METHOD FB_init : BOOL
VAR_INPUT
	bInitRetains : BOOL; // if TRUE, the retain variables are initialized (warm start / cold start)
	bInCopyCode : BOOL;  // if TRUE, the instance afterwards gets moved into the copy code (online change)
END_VAR
AddInput('aPoint1', aPoint1);
AddInput('aPoint2', aPoint2);
AddParameter('bNormalize', bNormalize);
AddInput('hrPrev', hrPrev);
AddOutput('aDirection', aDirection);
AddOutput('hresult',hresult);
END_METHOD

METHOD PUBLIC  Clone : I_Node
VAR
	pNode : POINTER TO Node_F_VN_PointToPointDirection_TcVnPoint2_DINT;
END_VAR
pNode := __NEW(Node_F_VN_PointToPointDirection_TcVnPoint2_DINT);
Clone := pNode^;
END_METHOD

METHOD PROTECTED OnExecute
hresult.Value := F_VN_PointToPointDirection_TcVnPoint2_DINT(
    aPoint1 := aPoint1.Value,
    aPoint2 := aPoint2.Value,
    aDirection := aDirection.Value,
    bNormalize := bNormalize.Value,
	hrPrev:= hrPrev.Value);
END_METHOD

METHOD PUBLIC PreExecutionCheck
VAR_INPUT
	Check : I_PreExecutionChecks;
END_VAR
END_METHOD

END_FUNCTION_BLOCK

// Nodes/Miscellaneous/Node_F_VN_PointToPointDirection_TcVnPoint2_LREAL
{attribute 'linkalways'} 
{attribute 'no_explicit_call' := 'This FB is a CLASS and must be accessed using methods or properties'}
{attribute 'enable_dynamic_creation'}
FUNCTION_BLOCK Node_F_VN_PointToPointDirection_TcVnPoint2_LREAL EXTENDS VisionNode
VAR
    aPoint1 : _TcVnPoint2_LREAL;
    aPoint2 : _TcVnPoint2_LREAL;
    aDirection : _TcVnVector2_LREAL;
    bNormalize : _BOOL(FALSE);
    hrPrev : _HRESULT(S_OK);
	hresult : _HRESULT(S_OK);
END_VAR

METHOD FB_init : BOOL
VAR_INPUT
	bInitRetains : BOOL; // if TRUE, the retain variables are initialized (warm start / cold start)
	bInCopyCode : BOOL;  // if TRUE, the instance afterwards gets moved into the copy code (online change)
END_VAR
AddInput('aPoint1', aPoint1);
AddInput('aPoint2', aPoint2);
AddParameter('bNormalize', bNormalize);
AddInput('hrPrev', hrPrev);
AddOutput('aDirection', aDirection);
AddOutput('hresult',hresult);
END_METHOD

METHOD PUBLIC  Clone : I_Node
VAR
	pNode : POINTER TO Node_F_VN_PointToPointDirection_TcVnPoint2_LREAL;
END_VAR
pNode := __NEW(Node_F_VN_PointToPointDirection_TcVnPoint2_LREAL);
Clone := pNode^;
END_METHOD

METHOD PROTECTED OnExecute
hresult.Value := F_VN_PointToPointDirection_TcVnPoint2_LREAL(
    aPoint1 := aPoint1.Value,
    aPoint2 := aPoint2.Value,
    aDirection := aDirection.Value,
    bNormalize := bNormalize.Value,
	hrPrev:= hrPrev.Value);
END_METHOD

METHOD PUBLIC PreExecutionCheck
VAR_INPUT
	Check : I_PreExecutionChecks;
END_VAR
END_METHOD

END_FUNCTION_BLOCK

// Nodes/Miscellaneous/Node_F_VN_PointToPointDirection_TcVnPoint2_REAL
{attribute 'linkalways'} 
{attribute 'no_explicit_call' := 'This FB is a CLASS and must be accessed using methods or properties'}
{attribute 'enable_dynamic_creation'}
FUNCTION_BLOCK Node_F_VN_PointToPointDirection_TcVnPoint2_REAL EXTENDS VisionNode
VAR
    aPoint1 : _TcVnPoint2_REAL;
    aPoint2 : _TcVnPoint2_REAL;
    aDirection : _TcVnVector2_REAL;
    bNormalize : _BOOL(FALSE);
    hrPrev : _HRESULT(S_OK);
	hresult : _HRESULT(S_OK);
END_VAR

METHOD FB_init : BOOL
VAR_INPUT
	bInitRetains : BOOL; // if TRUE, the retain variables are initialized (warm start / cold start)
	bInCopyCode : BOOL;  // if TRUE, the instance afterwards gets moved into the copy code (online change)
END_VAR
AddInput('aPoint1', aPoint1);
AddInput('aPoint2', aPoint2);
AddParameter('bNormalize', bNormalize);
AddInput('hrPrev', hrPrev);
AddOutput('aDirection', aDirection);
AddOutput('hresult',hresult);
END_METHOD

METHOD PUBLIC  Clone : I_Node
VAR
	pNode : POINTER TO Node_F_VN_PointToPointDirection_TcVnPoint2_REAL;
END_VAR
pNode := __NEW(Node_F_VN_PointToPointDirection_TcVnPoint2_REAL);
Clone := pNode^;
END_METHOD

METHOD PROTECTED OnExecute
hresult.Value := F_VN_PointToPointDirection_TcVnPoint2_REAL(
    aPoint1 := aPoint1.Value,
    aPoint2 := aPoint2.Value,
    aDirection := aDirection.Value,
    bNormalize := bNormalize.Value,
	hrPrev:= hrPrev.Value);
END_METHOD

METHOD PUBLIC PreExecutionCheck
VAR_INPUT
	Check : I_PreExecutionChecks;
END_VAR
END_METHOD

END_FUNCTION_BLOCK

// Nodes/Miscellaneous/Node_F_VN_PointToPointDistance_TcVnPoint2_DINT
{attribute 'linkalways'} 
{attribute 'no_explicit_call' := 'This FB is a CLASS and must be accessed using methods or properties'}
{attribute 'enable_dynamic_creation'}
FUNCTION_BLOCK Node_F_VN_PointToPointDistance_TcVnPoint2_DINT EXTENDS VisionNode
VAR
    aPoint1 : _TcVnPoint2_DINT;
    aPoint2 : _TcVnPoint2_DINT;
    fDistance : _LREAL(0.0);
    hrPrev : _HRESULT(S_OK);
	hresult : _HRESULT(S_OK);
END_VAR

METHOD FB_init : BOOL
VAR_INPUT
	bInitRetains : BOOL; // if TRUE, the retain variables are initialized (warm start / cold start)
	bInCopyCode : BOOL;  // if TRUE, the instance afterwards gets moved into the copy code (online change)
END_VAR
AddInput('aPoint1', aPoint1);
AddInput('aPoint2', aPoint2);
AddInput('hrPrev', hrPrev);
AddOutput('fDistance', fDistance);
AddOutput('hresult',hresult);
END_METHOD

METHOD PUBLIC  Clone : I_Node
VAR
	pNode : POINTER TO Node_F_VN_PointToPointDistance_TcVnPoint2_DINT;
END_VAR
pNode := __NEW(Node_F_VN_PointToPointDistance_TcVnPoint2_DINT);
Clone := pNode^;
END_METHOD

METHOD PROTECTED OnExecute
hresult.Value := F_VN_PointToPointDistance_TcVnPoint2_DINT(
    aPoint1 := aPoint1.Value,
    aPoint2 := aPoint2.Value,
    fDistance := fDistance.Value,
	hrPrev:= hrPrev.Value);
END_METHOD

METHOD PUBLIC PreExecutionCheck
VAR_INPUT
	Check : I_PreExecutionChecks;
END_VAR
END_METHOD

END_FUNCTION_BLOCK

// Nodes/Miscellaneous/Node_F_VN_PointToPointDistance_TcVnPoint2_LREAL
{attribute 'linkalways'} 
{attribute 'no_explicit_call' := 'This FB is a CLASS and must be accessed using methods or properties'}
{attribute 'enable_dynamic_creation'}
FUNCTION_BLOCK Node_F_VN_PointToPointDistance_TcVnPoint2_LREAL EXTENDS VisionNode
VAR
    aPoint1 : _TcVnPoint2_LREAL;
    aPoint2 : _TcVnPoint2_LREAL;
    fDistance : _LREAL(0.0);
    hrPrev : _HRESULT(S_OK);
	hresult : _HRESULT(S_OK);
END_VAR

METHOD FB_init : BOOL
VAR_INPUT
	bInitRetains : BOOL; // if TRUE, the retain variables are initialized (warm start / cold start)
	bInCopyCode : BOOL;  // if TRUE, the instance afterwards gets moved into the copy code (online change)
END_VAR
AddInput('aPoint1', aPoint1);
AddInput('aPoint2', aPoint2);
AddInput('hrPrev', hrPrev);
AddOutput('fDistance', fDistance);
AddOutput('hresult',hresult);
END_METHOD

METHOD PUBLIC  Clone : I_Node
VAR
	pNode : POINTER TO Node_F_VN_PointToPointDistance_TcVnPoint2_LREAL;
END_VAR
pNode := __NEW(Node_F_VN_PointToPointDistance_TcVnPoint2_LREAL);
Clone := pNode^;
END_METHOD

METHOD PROTECTED OnExecute
hresult.Value := F_VN_PointToPointDistance_TcVnPoint2_LREAL(
    aPoint1 := aPoint1.Value,
    aPoint2 := aPoint2.Value,
    fDistance := fDistance.Value,
	hrPrev:= hrPrev.Value);
END_METHOD

METHOD PUBLIC PreExecutionCheck
VAR_INPUT
	Check : I_PreExecutionChecks;
END_VAR
END_METHOD

END_FUNCTION_BLOCK

// Nodes/Miscellaneous/Node_F_VN_PointToPointDistance_TcVnPoint2_REAL
{attribute 'linkalways'} 
{attribute 'no_explicit_call' := 'This FB is a CLASS and must be accessed using methods or properties'}
{attribute 'enable_dynamic_creation'}
FUNCTION_BLOCK Node_F_VN_PointToPointDistance_TcVnPoint2_REAL EXTENDS VisionNode
VAR
    aPoint1 : _TcVnPoint2_REAL;
    aPoint2 : _TcVnPoint2_REAL;
    fDistance : _LREAL(0.0);
    hrPrev : _HRESULT(S_OK);
	hresult : _HRESULT(S_OK);
END_VAR

METHOD FB_init : BOOL
VAR_INPUT
	bInitRetains : BOOL; // if TRUE, the retain variables are initialized (warm start / cold start)
	bInCopyCode : BOOL;  // if TRUE, the instance afterwards gets moved into the copy code (online change)
END_VAR
AddInput('aPoint1', aPoint1);
AddInput('aPoint2', aPoint2);
AddInput('hrPrev', hrPrev);
AddOutput('fDistance', fDistance);
AddOutput('hresult',hresult);
END_METHOD

METHOD PUBLIC  Clone : I_Node
VAR
	pNode : POINTER TO Node_F_VN_PointToPointDistance_TcVnPoint2_REAL;
END_VAR
pNode := __NEW(Node_F_VN_PointToPointDistance_TcVnPoint2_REAL);
Clone := pNode^;
END_METHOD

METHOD PROTECTED OnExecute
hresult.Value := F_VN_PointToPointDistance_TcVnPoint2_REAL(
    aPoint1 := aPoint1.Value,
    aPoint2 := aPoint2.Value,
    fDistance := fDistance.Value,
	hrPrev:= hrPrev.Value);
END_METHOD

METHOD PUBLIC PreExecutionCheck
VAR_INPUT
	Check : I_PreExecutionChecks;
END_VAR
END_METHOD

END_FUNCTION_BLOCK

// Nodes/Miscellaneous/Node_F_VN_RotatedRectangleCorners
{attribute 'linkalways'} 
{attribute 'no_explicit_call' := 'This FB is a CLASS and must be accessed using methods or properties'}
{attribute 'enable_dynamic_creation'}
FUNCTION_BLOCK Node_F_VN_RotatedRectangleCorners EXTENDS VisionNode
VAR
    stRect : _TcVnRotatedRectangle;
    aCorners : _TcVnArray4_Point2_REAL;
    hrPrev : _HRESULT(S_OK);
	hresult : _HRESULT(S_OK);
END_VAR

METHOD FB_init : BOOL
VAR_INPUT
	bInitRetains : BOOL; // if TRUE, the retain variables are initialized (warm start / cold start)
	bInCopyCode : BOOL;  // if TRUE, the instance afterwards gets moved into the copy code (online change)
END_VAR
AddInput('stRect', stRect);
AddInput('hrPrev', hrPrev);
AddOutput('aCorners', aCorners);
AddOutput('hresult',hresult);
END_METHOD

METHOD PUBLIC  Clone : I_Node
VAR
	pNode : POINTER TO Node_F_VN_RotatedRectangleCorners;
END_VAR
pNode := __NEW(Node_F_VN_RotatedRectangleCorners);
Clone := pNode^;
END_METHOD

METHOD PROTECTED OnExecute
hresult.Value := F_VN_RotatedRectangleCorners(
    stRect := stRect.Value,
    aCorners := aCorners.Value,
	hrPrev:= hrPrev.Value);
END_METHOD

METHOD PUBLIC PreExecutionCheck
VAR_INPUT
	Check : I_PreExecutionChecks;
END_VAR
END_METHOD

END_FUNCTION_BLOCK

// Nodes/Miscellaneous/Node_F_VN_RotatedRectangleIntersection
{attribute 'linkalways'} 
{attribute 'no_explicit_call' := 'This FB is a CLASS and must be accessed using methods or properties'}
{attribute 'enable_dynamic_creation'}
FUNCTION_BLOCK Node_F_VN_RotatedRectangleIntersection EXTENDS VisionNode
VAR
    stRect1 : _TcVnRotatedRectangle;
    stRect2 : _TcVnRotatedRectangle;
    ipIntersection : _ITcVnContainer;
    eIntersection : _ETcVnRectangleIntersection(ETcVnRectangleIntersection.TCVN_RI_NONE);
    hrPrev : _HRESULT(S_OK);
	hresult : _HRESULT(S_OK);
END_VAR

METHOD FB_init : BOOL
VAR_INPUT
	bInitRetains : BOOL; // if TRUE, the retain variables are initialized (warm start / cold start)
	bInCopyCode : BOOL;  // if TRUE, the instance afterwards gets moved into the copy code (online change)
END_VAR
AddInput('stRect1', stRect1);
AddInput('stRect2', stRect2);
AddInput('hrPrev', hrPrev);
AddOutput('ipIntersection', ipIntersection);
AddOutput('eIntersection', eIntersection);
AddOutput('hresult',hresult);
END_METHOD

METHOD PUBLIC  Clone : I_Node
VAR
	pNode : POINTER TO Node_F_VN_RotatedRectangleIntersection;
END_VAR
pNode := __NEW(Node_F_VN_RotatedRectangleIntersection);
Clone := pNode^;
END_METHOD

METHOD PROTECTED OnExecute
VAR
    intersection : ETcVnRectangleIntersection;
END_VAR
hresult.Value := F_VN_RotatedRectangleIntersection(
    stRect1 := stRect1.Value,
    stRect2 := stRect2.Value,
    ipIntersection := ipIntersection.Value,
    eIntersection := intersection,
	hrPrev:= hrPrev.Value);

 eIntersection.Value := intersection;
END_METHOD

METHOD PUBLIC PreExecutionCheck
VAR_INPUT
	Check : I_PreExecutionChecks;
END_VAR
END_METHOD

END_FUNCTION_BLOCK

// Nodes/Neural Network/Node_F_VN_Reduce
{attribute 'linkalways'} 
{attribute 'no_explicit_call' := 'This FB is a CLASS and must be accessed using methods or properties'}
{attribute 'enable_dynamic_creation'}
FUNCTION_BLOCK Node_F_VN_Reduce EXTENDS VisionNode
VAR
    ipSrcImage : _ITcVnImage;
    ipDestImage : _ITcVnImage;
	nDim : _DINT(0);
	eReduceType : _ETcVnReduceType(ETcVnReduceType.TCVN_RT_REDUCE_AVG);
    hrPrev : _HRESULT(S_OK);
	hresult : _HRESULT(S_OK);
END_VAR

METHOD FB_init : BOOL
VAR_INPUT
	bInitRetains : BOOL; // if TRUE, the retain variables are initialized (warm start / cold start)
	bInCopyCode : BOOL;  // if TRUE, the instance afterwards gets moved into the copy code (online change)
END_VAR
AddInput('ipSrcImage', ipSrcImage);
AddInput('hrPrev', hrPrev);
AddParameter('nDim', nDim);
AddParameter('eReduceType', eReduceType);
AddOutput('ipDestImage', ipDestImage);
AddOutput('hresult',hresult);
END_METHOD

METHOD PUBLIC  Clone : I_Node
VAR
	pNode : POINTER TO Node_F_VN_Reduce;
END_VAR
pNode := __NEW(Node_F_VN_Reduce);
Clone := pNode^;
END_METHOD

METHOD PROTECTED OnExecute
hresult.Value := F_VN_Reduce(
	ipSrcImage := ipSrcImage.Value,
	ipDestImage := ipDestImage.Value,
	nDim := nDim.Value,
	eReduceType := eReduceType.Value,
	hrPrev:= hrPrev.Value);
END_METHOD

METHOD PUBLIC PreExecutionCheck
VAR_INPUT
	Check : I_PreExecutionChecks;
END_VAR
VAR
	nDimValue : DINT;
END_VAR
Check.IsTrue(ipSrcImage.IsValid, 'ipSrcImage must contain an image');
Check.IsTrue(ipSrcImage.HasChannelCount(1), 'ipSrcImage must have 1 channel');
Check.IsTrue(ipSrcImage.IsElementType(ETcVnElementType.TCVN_ET_USINT) OR_ELSE ipSrcImage.IsElementType(ETcVnElementType.TCVN_ET_REAL), 'ipSrcImage must have 32 bit pixel depth');

nDimValue := nDim.Value;
Check.IsTrue(nDimValue = 0 OR_ELSE nDimValue = 1 OR_ELSE nDimValue = 2, 'nDim must be 0, 1 or 2');
END_METHOD

END_FUNCTION_BLOCK

// Nodes/Neural Network/Node_F_VN_ReduceArg
{attribute 'linkalways'} 
{attribute 'no_explicit_call' := 'This FB is a CLASS and must be accessed using methods or properties'}
{attribute 'enable_dynamic_creation'}
FUNCTION_BLOCK Node_F_VN_ReduceArg EXTENDS VisionNode
VAR
    ipSrcImage : _ITcVnImage;
    ipDestImage : _ITcVnImage;
	nDim : _DINT(0);
	eReduceType : _DINT(0);
    hrPrev : _HRESULT(S_OK);
	hresult : _HRESULT(S_OK);
END_VAR

METHOD FB_init : BOOL
VAR_INPUT
	bInitRetains : BOOL; // if TRUE, the retain variables are initialized (warm start / cold start)
	bInCopyCode : BOOL;  // if TRUE, the instance afterwards gets moved into the copy code (online change)
END_VAR
AddInput('ipSrcImage', ipSrcImage);
AddInput('hrPrev', hrPrev);
AddParameter('nDim', nDim);
AddParameter('eReduceType', eReduceType);
AddOutput('ipDestImage', ipDestImage);
AddOutput('hresult',hresult);
END_METHOD

METHOD PUBLIC  Clone : I_Node
VAR
	pNode : POINTER TO Node_F_VN_ReduceArg;
END_VAR
pNode := __NEW(Node_F_VN_ReduceArg);
Clone := pNode^;
END_METHOD

METHOD PROTECTED OnExecute
hresult.Value := F_VN_ReduceArg(
	ipSrcImage := ipSrcImage.Value,
	ipDestImage := ipDestImage.Value,
	nDim := nDim.Value,
	eReduceType := eReduceType.Value,
	hrPrev:= hrPrev.Value);
END_METHOD

METHOD PUBLIC PreExecutionCheck
VAR_INPUT
	Check : I_PreExecutionChecks;
END_VAR
VAR
	nDimValue : DINT;
END_VAR
Check.IsTrue(ipSrcImage.IsValid, 'ipSrcImage must contain an image');
// Check.IsTrue(ipSrcImage.HasChannelCount(1), 'ipSrcImage must have 1 channel');
// Check.IsTrue(ipSrcImage.IsElementType(ETcVnElementType.TCVN_ET_USINT) OR_ELSE ipSrcImage.IsElementType(ETcVnElementType.TCVN_ET_REAL), 'ipSrcImage must have 32 bit pixel depth');

nDimValue := nDim.Value;
Check.IsTrue(nDimValue = 0 OR_ELSE nDimValue = 1 OR_ELSE nDimValue = 2, 'nDim must be 0, 1 or 2');
END_METHOD

END_FUNCTION_BLOCK

// Nodes/Neural Network/Node_F_VN_Sigmoid
{attribute 'linkalways'} 
{attribute 'no_explicit_call' := 'This FB is a CLASS and must be accessed using methods or properties'}
{attribute 'enable_dynamic_creation'}
FUNCTION_BLOCK Node_F_VN_Sigmoid EXTENDS VisionNode
VAR
    ipSrcImage : _ITcVnImage;
    ipDestImage : _ITcVnImage;
    hrPrev : _HRESULT(S_OK);
	hresult : _HRESULT(S_OK);
END_VAR

METHOD FB_init : BOOL
VAR_INPUT
	bInitRetains : BOOL; // if TRUE, the retain variables are initialized (warm start / cold start)
	bInCopyCode : BOOL;  // if TRUE, the instance afterwards gets moved into the copy code (online change)
END_VAR
AddInput('ipSrcImage', ipSrcImage);
AddInput('hrPrev', hrPrev);
AddOutput('ipDestImage', ipDestImage);
AddOutput('hresult',hresult);
END_METHOD

METHOD PUBLIC  Clone : I_Node
VAR
	pNode : POINTER TO Node_F_VN_Sigmoid;
END_VAR
pNode := __NEW(Node_F_VN_Sigmoid);
Clone := pNode^;
END_METHOD

METHOD PROTECTED OnExecute
hresult.Value := F_VN_Sigmoid(
    ipSrcImage := ipSrcImage.Value,
	ipDestImage := ipDestImage.Value,
	hrPrev:= hrPrev.Value);
END_METHOD

METHOD PUBLIC PreExecutionCheck
VAR_INPUT
	Check : I_PreExecutionChecks;
END_VAR
Check.IsTrue(ipSrcImage.IsValid, 'ipSrcImage must contain an image');
Check.IsTrue(ipSrcImage.IsElementType(ETcVnElementType.TCVN_ET_REAL), 'ipSrcImage must be element type REAL');
END_METHOD

END_FUNCTION_BLOCK

// Nodes/Neural Network/Node_F_VN_SigmoidExp
{attribute 'linkalways'} 
{attribute 'no_explicit_call' := 'This FB is a CLASS and must be accessed using methods or properties'}
{attribute 'enable_dynamic_creation'}
FUNCTION_BLOCK Node_F_VN_SigmoidExp EXTENDS VisionNode
VAR
    ipSrcImage : _ITcVnImage;
    ipDestImage : _ITcVnImage;
    fShift : _REAL(0.0);
    fSteepness : _REAL(0.0);
    hrPrev : _HRESULT(S_OK);
	hresult : _HRESULT(S_OK);
END_VAR

METHOD FB_init : BOOL
VAR_INPUT
	bInitRetains : BOOL; // if TRUE, the retain variables are initialized (warm start / cold start)
	bInCopyCode : BOOL;  // if TRUE, the instance afterwards gets moved into the copy code (online change)
END_VAR
AddInput('ipSrcImage', ipSrcImage);
AddParameter('fShift', fShift);
AddParameter('fSteepness', fSteepness);
AddInput('hrPrev', hrPrev);
AddOutput('ipDestImage', ipDestImage);
AddOutput('hresult',hresult);
END_METHOD

METHOD PUBLIC  Clone : I_Node
VAR
	pNode : POINTER TO Node_F_VN_SigmoidExp;
END_VAR
pNode := __NEW(Node_F_VN_SigmoidExp);
Clone := pNode^;
END_METHOD

METHOD PROTECTED OnExecute
hresult.Value := F_VN_SigmoidExp(
    ipSrcImage := ipSrcImage.Value,
	ipDestImage := ipDestImage.Value,
    fShift := fShift.Value,
    fSteepness := fSteepness.Value,
	hrPrev:= hrPrev.Value);
END_METHOD

METHOD PUBLIC PreExecutionCheck
VAR_INPUT
	Check : I_PreExecutionChecks;
END_VAR
Check.IsTrue(ipSrcImage.IsValid, 'ipSrcImage must contain an image');
Check.IsTrue(ipSrcImage.IsElementType(ETcVnElementType.TCVN_ET_REAL), 'ipSrcImage must be element type REAL');
END_METHOD

END_FUNCTION_BLOCK

// Nodes/Neural Network/Node_F_VN_SoftMax
{attribute 'linkalways'} 
{attribute 'no_explicit_call' := 'This FB is a CLASS and must be accessed using methods or properties'}
{attribute 'enable_dynamic_creation'}
FUNCTION_BLOCK Node_F_VN_SoftMax EXTENDS VisionNode
VAR
    ipSrcImage : _ITcVnImage;
    ipDestImage : _ITcVnImage;
    bFlatten : _BOOL(FALSE);
    hrPrev : _HRESULT(S_OK);
	hresult : _HRESULT(S_OK);
END_VAR

METHOD FB_init : BOOL
VAR_INPUT
	bInitRetains : BOOL; // if TRUE, the retain variables are initialized (warm start / cold start)
	bInCopyCode : BOOL;  // if TRUE, the instance afterwards gets moved into the copy code (online change)
END_VAR
AddInput('ipSrcImage', ipSrcImage);
AddParameter('bFlatten', bFlatten);
AddInput('hrPrev', hrPrev);
AddOutput('ipDestImage', ipDestImage);
AddOutput('hresult',hresult);
END_METHOD

METHOD PUBLIC  Clone : I_Node
VAR
	pNode : POINTER TO Node_F_VN_SoftMax;
END_VAR
pNode := __NEW(Node_F_VN_SoftMax);
Clone := pNode^;
END_METHOD

METHOD PROTECTED OnExecute
hresult.Value := F_VN_SoftMax(
    ipSrcImage := ipSrcImage.Value,
	ipDestImage := ipDestImage.Value,
    bFlatten := bFlatten.Value,
	hrPrev:= hrPrev.Value);
END_METHOD

METHOD PUBLIC PreExecutionCheck
VAR_INPUT
	Check : I_PreExecutionChecks;
END_VAR
Check.IsTrue(ipSrcImage.IsValid, 'ipSrcImage must contain an image');
Check.IsTrue(ipSrcImage.IsElementType(ETcVnElementType.TCVN_ET_REAL), 'ipSrcImage must be element type REAL');
Check.IsTrue(ipSrcImage.HasChannelCount(1), 'ipSrcImage must have 1 channel');
END_METHOD

END_FUNCTION_BLOCK

// Nodes/OCR/Node_F_VN_OCR
{attribute 'linkalways'} 
{attribute 'no_explicit_call' := 'This FB is a CLASS and must be accessed using methods or properties'}
{attribute 'enable_dynamic_creation'}
FUNCTION_BLOCK Node_F_VN_OCR EXTENDS VisionNode
VAR
	ipSrcImage : _ITcVnImage;
    eModel : _ETcVnOcrModelType(ETcVnOcrModelType.TCVN_OMT_NUMBERS);
    ipCharacters : _ITcVnContainer;
    hrPrev : _HRESULT(S_OK);
	hresult : _HRESULT(S_OK);
END_VAR

METHOD FB_init : BOOL
VAR_INPUT
	bInitRetains : BOOL; // if TRUE, the retain variables are initialized (warm start / cold start)
	bInCopyCode : BOOL;  // if TRUE, the instance afterwards gets moved into the copy code (online change)
END_VAR
AddInput('ipSrcImage', ipSrcImage);
AddParameter('eModel', eModel);
AddInput('hrPrev', hrPrev);
AddOutput('ipCharacters', ipCharacters);
AddOutput('hresult',hresult);
END_METHOD

METHOD PUBLIC  Clone : I_Node
VAR
	pNode : POINTER TO Node_F_VN_OCR;
END_VAR
pNode := __NEW(Node_F_VN_OCR);
Clone := pNode^;
END_METHOD

METHOD PROTECTED OnExecute
hresult.Value := F_VN_OCR(
	ipSrcImage := ipSrcImage.Value,
    eModel := eModel.Value,
	ipCharacters := ipCharacters.Value,
	hrPrev:= hrPrev.Value);
END_METHOD

METHOD PUBLIC PreExecutionCheck
VAR_INPUT
	Check : I_PreExecutionChecks;
END_VAR
VAR
    result : HRESULT;
END_VAR
result := F_VN_CheckFunctionInitialization(ETcVnInitializableFunction.TCVN_IF_OCR, eModel.Value, S_OK);
Check.IsTrue((result = S_OK), 'Invalid OCR model');

Check.IsTrue(ipSrcImage.IsValid, 'ipSrcImage must contain an image');
Check.IsTrue(ipSrcImage.IsPixelDepth(8), 'ipSrcImage must have 8 bit pixel depth');
Check.IsTrue(ipSrcImage.HasChannelCount(1), 'ipSrcImage must contain 1 channel');
END_METHOD

END_FUNCTION_BLOCK

// Nodes/OCR/Node_F_VN_OCRExp
{attribute 'linkalways'} 
{attribute 'no_explicit_call' := 'This FB is a CLASS and must be accessed using methods or properties'}
{attribute 'enable_dynamic_creation'}
FUNCTION_BLOCK Node_F_VN_OCRExp EXTENDS VisionNode
VAR
	ipSrcImage : _ITcVnImage;
    eModel : _ETcVnOcrModelType(ETcVnOcrModelType.TCVN_OMT_NUMBERS);
    ipCharacters : _ITcVnContainer;
    sPattern : _STRING('');
    eOcrOptions : _ETcVnOcrOptions(ETcVnOcrOptions.TCVN_OO_NONE);
    ipBoundingBoxes : _ITcVnContainer;
    ipConfidences : _ITcVnContainer;
    hrPrev : _HRESULT(S_OK);
    fMinConfidence : _REAL(0.0);
	hresult : _HRESULT(S_OK);
END_VAR

METHOD FB_init : BOOL
VAR_INPUT
	bInitRetains : BOOL; // if TRUE, the retain variables are initialized (warm start / cold start)
	bInCopyCode : BOOL;  // if TRUE, the instance afterwards gets moved into the copy code (online change)
END_VAR
AddInput('ipSrcImage', ipSrcImage);
AddParameter('eModel', eModel);
AddParameter('sPattern', sPattern);
AddParameter('eOcrOptions', eOcrOptions);
AddInput('hrPrev', hrPrev);
AddOutput('ipCharacters', ipCharacters);
AddOutput('ipBoundingBoxes', ipBoundingBoxes);
AddOutput('ipConfidences', ipConfidences);
AddOutput('fMinConfidence', fMinConfidence);
AddOutput('hresult',hresult);
END_METHOD

METHOD PUBLIC  Clone : I_Node
VAR
	pNode : POINTER TO Node_F_VN_OCRExp;
END_VAR
pNode := __NEW(Node_F_VN_OCRExp);
Clone := pNode^;
END_METHOD

METHOD PROTECTED OnExecute
VAR
    minConfidence : REAL;
END_VAR
hresult.Value := F_VN_OCRExp(
	ipSrcImage := ipSrcImage.Value,
    eModel := eModel.Value,
	ipCharacters := ipCharacters.Value,
    sPattern := sPattern.Value,
    eOcrOptions := eOcrOptions.Value,
    ipBoundingBoxes := ipBoundingBoxes.Value,
    ipConfidences := ipConfidences.Value,
	hrPrev := hrPrev.Value,
    fMinConfidence => minConfidence);

fMinConfidence.Value := minConfidence;
END_METHOD

METHOD PUBLIC PreExecutionCheck
VAR_INPUT
	Check : I_PreExecutionChecks;
END_VAR
VAR
    result : HRESULT;
END_VAR
result := F_VN_CheckFunctionInitialization(ETcVnInitializableFunction.TCVN_IF_OCR, eModel.Value, S_OK);
Check.IsTrue((result = S_OK), 'Invalid OCR model');

Check.IsTrue(ipSrcImage.IsValid, 'ipSrcImage must contain an image');
Check.IsTrue(ipSrcImage.IsPixelDepth(8), 'ipSrcImage must have 8 bit pixel depth');
Check.IsTrue(ipSrcImage.HasChannelCount(1), 'ipSrcImage must contain 1 channel');
END_METHOD

END_FUNCTION_BLOCK

// Nodes/Polarization/Node_F_VN_AngleAndDegreeOfLinearPolarization
{attribute 'linkalways'}
{attribute 'no_explicit_call' := 'This FB is a CLASS and must be accessed using methods or properties'}
{attribute 'enable_dynamic_creation'}
FUNCTION_BLOCK Node_F_VN_AngleAndDegreeOfLinearPolarization EXTENDS VisionNode
VAR
    ip0Deg : _ITcVnImage;
    ip45Deg : _ITcVnImage;
    ip90Deg : _ITcVnImage;
    ip135Deg : _ITcVnImage;
    ipAoLP : _ITcVnImage;
    ipDoLP : _ITcVnImage;
    eDestType : _ETcVnElementType(ETcVnElementType.TCVN_ET_REAL);
    hrPrev : _HRESULT(S_OK);
    hresult : _HRESULT(S_OK);
END_VAR

METHOD FB_init : BOOL
VAR_INPUT
    bInitRetains : BOOL;
    bInCopyCode : BOOL;
END_VAR
AddInput('ip0Deg', ip0Deg);
AddInput('ip45Deg', ip45Deg);
AddInput('ip90Deg', ip90Deg);
AddInput('ip135Deg', ip135Deg);
AddOutput('ipAoLP', ipAoLP);
AddOutput('ipDoLP', ipDoLP);
AddParameter('eDestType', eDestType);
AddInput('hrPrev', hrPrev);
AddOutput('hresult', hresult);
END_METHOD

METHOD PUBLIC Clone : I_Node
VAR
    pNode : POINTER TO Node_F_VN_AngleAndDegreeOfLinearPolarization;
END_VAR
pNode := __NEW(Node_F_VN_AngleAndDegreeOfLinearPolarization);
Clone := pNode^;
END_METHOD

METHOD PROTECTED OnExecute
hresult.Value := F_VN_AngleAndDegreeOfLinearPolarization(
    ip0Deg := ip0Deg.Value,
    ip45Deg := ip45Deg.Value,
    ip90Deg := ip90Deg.Value,
    ip135Deg := ip135Deg.Value,
    ipAoLP := ipAoLP.Value,
    ipDoLP := ipDoLP.Value,
    eDestType := eDestType.Value,
    hrPrev := hrPrev.Value);
END_METHOD

METHOD PUBLIC PreExecutionCheck
VAR_INPUT
    Check : I_PreExecutionChecks;
END_VAR
Check.IsTrue(ip0Deg.IsValid, 'ip0Deg must contain an image');
Check.IsTrue(ip0Deg.IsElementType(ETcVnElementType.TCVN_ET_USINT) OR
             ip0Deg.IsElementType(ETcVnElementType.TCVN_ET_UINT), 'Polarization components must contain USINT or UINT elements');
Check.IsTrue(ip0Deg.HasChannelCount(1) OR ip0Deg.HasChannelCount(3), 'Polarization components must contain 1 or 3 channels');
Check.IsTrue(ip45Deg.IsValid, 'ip45Deg must contain an image');
Check.IsTrue(ImagesHaveMatchingPixelFormats(ip0Deg.Value, ip45Deg.Value), 'Source images must have matching pixel formats');
Check.IsTrue(IsImage1SizeEqualToImage2Size(ip0Deg.Value, ip45Deg.Value), 'Source images must have matching dimensions');
Check.IsTrue(ip90Deg.IsValid, 'ip90Deg must contain an image');
Check.IsTrue(ImagesHaveMatchingPixelFormats(ip0Deg.Value, ip90Deg.Value), 'Source images must have matching pixel formats');
Check.IsTrue(IsImage1SizeEqualToImage2Size(ip0Deg.Value, ip90Deg.Value), 'Source images must have matching dimensions');
Check.IsTrue(ip135Deg.IsValid, 'ip135Deg must contain an image');
Check.IsTrue(ImagesHaveMatchingPixelFormats(ip0Deg.Value, ip135Deg.Value), 'Source images must have matching pixel formats');
Check.IsTrue(IsImage1SizeEqualToImage2Size(ip0Deg.Value, ip135Deg.Value), 'Source images must have matching dimensions');
Check.IsTrue((eDestType.Value = ETcVnElementType.TCVN_ET_REAL) OR
             (eDestType.Value = ETcVnElementType.TCVN_ET_USINT), 'Unsupported eDestType');
Check.IsTrue((ipAoLP.Value = 0) OR ((ipAoLP.Value <> ip0Deg.Value) AND
             (ipAoLP.Value <> ip45Deg.Value) AND
             (ipAoLP.Value <> ip90Deg.Value) AND
             (ipAoLP.Value <> ip135Deg.Value)), 'ipAoLP must be different from the source images');
Check.IsTrue((ipDoLP.Value = 0) OR ((ipDoLP.Value <> ip0Deg.Value) AND
             (ipDoLP.Value <> ip45Deg.Value) AND
             (ipDoLP.Value <> ip90Deg.Value) AND
             (ipDoLP.Value <> ip135Deg.Value)), 'ipDoLP must be different from the source images');
END_METHOD

END_FUNCTION_BLOCK

// Nodes/Polarization/Node_F_VN_DemosaicPolarizedImage
{attribute 'linkalways'}
{attribute 'no_explicit_call' := 'This FB is a CLASS and must be accessed using methods or properties'}
{attribute 'enable_dynamic_creation'}
FUNCTION_BLOCK Node_F_VN_DemosaicPolarizedImage EXTENDS VisionNode
VAR
    ipPolarizedImage : _ITcVnImage;
    ip0Deg : _ITcVnImage;
    ip45Deg : _ITcVnImage;
    ip90Deg : _ITcVnImage;
    ip135Deg : _ITcVnImage;
    eEncoding : _ETcVnPixelEncoding(ETcVnPixelEncoding.TCVN_PE_NONE);
    eInterpolation : _ETcVnPolarizedImageInterpolation(ETcVnPolarizedImageInterpolation.TCVN_PII_NONE);
    hrPrev : _HRESULT(S_OK);
    hresult : _HRESULT(S_OK);
END_VAR

METHOD FB_init : BOOL
VAR_INPUT
    bInitRetains : BOOL;
    bInCopyCode : BOOL;
END_VAR
AddInput('ipPolarizedImage', ipPolarizedImage);
AddOutput('ip0Deg', ip0Deg);
AddOutput('ip45Deg', ip45Deg);
AddOutput('ip90Deg', ip90Deg);
AddOutput('ip135Deg', ip135Deg);
AddParameter('eEncoding', eEncoding);
AddParameter('eInterpolation', eInterpolation);
AddInput('hrPrev', hrPrev);
AddOutput('hresult', hresult);
END_METHOD

METHOD PUBLIC Clone : I_Node
VAR
    pNode : POINTER TO Node_F_VN_DemosaicPolarizedImage;
END_VAR
pNode := __NEW(Node_F_VN_DemosaicPolarizedImage);
Clone := pNode^;
END_METHOD

METHOD PROTECTED OnExecute
hresult.Value := F_VN_DemosaicPolarizedImage(
    ipPolarizedImage := ipPolarizedImage.Value,
    ip0Deg := ip0Deg.Value,
    ip45Deg := ip45Deg.Value,
    ip90Deg := ip90Deg.Value,
    ip135Deg := ip135Deg.Value,
    eEncoding := eEncoding.Value,
    eInterpolation := eInterpolation.Value,
    hrPrev := hrPrev.Value);
END_METHOD

METHOD PUBLIC PreExecutionCheck
VAR_INPUT
    Check : I_PreExecutionChecks;
END_VAR
Check.IsTrue(ipPolarizedImage.IsValid, 'ipPolarizedImage must contain an image');
Check.IsTrue(ipPolarizedImage.IsElementType(ETcVnElementType.TCVN_ET_USINT) OR
             ipPolarizedImage.IsElementType(ETcVnElementType.TCVN_ET_UINT), 'Polarized image must contain USINT or UINT elements');
Check.IsTrue((eEncoding.Value = ETcVnPixelEncoding.TCVN_PE_NONE) OR
             (eEncoding.Value = ETcVnPixelEncoding.TCVN_PE_BAYER_GR) OR
             (eEncoding.Value = ETcVnPixelEncoding.TCVN_PE_BAYER_RG) OR
             (eEncoding.Value = ETcVnPixelEncoding.TCVN_PE_BAYER_GB) OR
             (eEncoding.Value = ETcVnPixelEncoding.TCVN_PE_BAYER_BG), 'Unsupported eEncoding');
Check.IsTrue((eInterpolation.Value = ETcVnPolarizedImageInterpolation.TCVN_PII_NONE) OR
             (eInterpolation.Value = ETcVnPolarizedImageInterpolation.TCVN_PII_NEAREST_NEIGHBOR) OR
             (eInterpolation.Value = ETcVnPolarizedImageInterpolation.TCVN_PII_BILINEAR) OR
             (eInterpolation.Value = ETcVnPolarizedImageInterpolation.TCVN_PII_BICUBIC) OR
             (eInterpolation.Value = ETcVnPolarizedImageInterpolation.TCVN_PII_LANCZOS4), 'Unsupported eInterpolation');
Check.IsTrue((ip0Deg.Value = 0) OR (ip0Deg.Value <> ipPolarizedImage.Value), 'ip0Deg must be different from the source image');
Check.IsTrue((ip45Deg.Value = 0) OR (ip45Deg.Value <> ipPolarizedImage.Value), 'ip45Deg must be different from the source image');
Check.IsTrue((ip90Deg.Value = 0) OR (ip90Deg.Value <> ipPolarizedImage.Value), 'ip90Deg must be different from the source image');
Check.IsTrue((ip135Deg.Value = 0) OR (ip135Deg.Value <> ipPolarizedImage.Value), 'ip135Deg must be different from the source image');
END_METHOD

END_FUNCTION_BLOCK

// Nodes/Polarization/Node_F_VN_PolarizedImageGlareReduction
{attribute 'linkalways'}
{attribute 'no_explicit_call' := 'This FB is a CLASS and must be accessed using methods or properties'}
{attribute 'enable_dynamic_creation'}
FUNCTION_BLOCK Node_F_VN_PolarizedImageGlareReduction EXTENDS VisionNode
VAR
    ipPolarizedImage : _ITcVnImage;
    ipDestImage : _ITcVnImage;
    eEncoding : _ETcVnPixelEncoding(ETcVnPixelEncoding.TCVN_PE_NONE);
    fIndex : _REAL(0.0);
    hrPrev : _HRESULT(S_OK);
    hresult : _HRESULT(S_OK);
END_VAR

METHOD FB_init : BOOL
VAR_INPUT
    bInitRetains : BOOL;
    bInCopyCode : BOOL;
END_VAR
AddInput('ipPolarizedImage', ipPolarizedImage);
AddOutput('ipDestImage', ipDestImage);
AddParameter('eEncoding', eEncoding);
AddParameter('fIndex', fIndex);
AddInput('hrPrev', hrPrev);
AddOutput('hresult', hresult);
END_METHOD

METHOD PUBLIC Clone : I_Node
VAR
    pNode : POINTER TO Node_F_VN_PolarizedImageGlareReduction;
END_VAR
pNode := __NEW(Node_F_VN_PolarizedImageGlareReduction);
Clone := pNode^;
END_METHOD

METHOD PROTECTED OnExecute
hresult.Value := F_VN_PolarizedImageGlareReduction(
    ipPolarizedImage := ipPolarizedImage.Value,
    ipDestImage := ipDestImage.Value,
    eEncoding := eEncoding.Value,
    fIndex := fIndex.Value,
    hrPrev := hrPrev.Value);
END_METHOD

METHOD PUBLIC PreExecutionCheck
VAR_INPUT
    Check : I_PreExecutionChecks;
END_VAR
Check.IsTrue(ipPolarizedImage.IsValid, 'ipPolarizedImage must contain an image');
Check.IsTrue(ipPolarizedImage.IsElementType(ETcVnElementType.TCVN_ET_USINT) OR
             ipPolarizedImage.IsElementType(ETcVnElementType.TCVN_ET_UINT), 'Polarized image must contain USINT or UINT elements');
Check.IsTrue((eEncoding.Value = ETcVnPixelEncoding.TCVN_PE_NONE) OR
             (eEncoding.Value = ETcVnPixelEncoding.TCVN_PE_BAYER_GR) OR
             (eEncoding.Value = ETcVnPixelEncoding.TCVN_PE_BAYER_RG) OR
             (eEncoding.Value = ETcVnPixelEncoding.TCVN_PE_BAYER_GB) OR
             (eEncoding.Value = ETcVnPixelEncoding.TCVN_PE_BAYER_BG), 'Unsupported eEncoding');
Check.IsTrue((fIndex.Value >= 0.0) AND (fIndex.Value <= 3.0), 'Intensity index must be between 0 and 3');
END_METHOD

END_FUNCTION_BLOCK

// Nodes/Texture Analysis/Node_F_VN_Granulometry
{attribute 'linkalways'} 
{attribute 'no_explicit_call' := 'This FB is a CLASS and must be accessed using methods or properties'}
{attribute 'enable_dynamic_creation'}
FUNCTION_BLOCK Node_F_VN_Granulometry EXTENDS VisionNode
VAR
    ipImage : _ITcVnImage;
    ipIntensityDiffs : _ITcVnContainer;
    eMorphType : _ETcVnMorphologicalOperator(ETcVnMorphologicalOperator.TCVN_MO_CLOSING);
    nMinSize : _UDINT(3);
    nMaxSize : _UDINT(3);
    nStep : _UDINT(2);
    hrPrev : _HRESULT(S_OK);
	hresult : _HRESULT(S_OK);
END_VAR

METHOD FB_init : BOOL
VAR_INPUT
	bInitRetains : BOOL; // if TRUE, the retain variables are initialized (warm start / cold start)
	bInCopyCode : BOOL;  // if TRUE, the instance afterwards gets moved into the copy code (online change)
END_VAR
AddInput('ipImage', ipImage);
AddParameter('eMorphType', eMorphType);
AddParameter('nMinSize', nMinSize);
AddParameter('nMaxSize', nMaxSize);
AddParameter('nStep', nStep);
AddInput('hrPrev', hrPrev);
AddOutput('ipIntensityDiffs', ipIntensityDiffs);
AddOutput('hresult',hresult);
END_METHOD

METHOD PUBLIC  Clone : I_Node
VAR
	pNode : POINTER TO Node_F_VN_Granulometry;
END_VAR
pNode := __NEW(Node_F_VN_Granulometry);
Clone := pNode^;
END_METHOD

METHOD PROTECTED OnExecute
hresult.Value := F_VN_Granulometry(
    ipImage := ipImage.Value,
    ipIntensityDiffs := ipIntensityDiffs.Value,
    eMorphType := eMorphType.Value,
    nMinSize := nMinSize.Value,
    nMaxSize := nMaxSize.Value,
    nStep := nStep.Value,
	hrPrev:= hrPrev.Value);
END_METHOD

METHOD PUBLIC PreExecutionCheck
VAR_INPUT
	Check : I_PreExecutionChecks;
END_VAR
Check.IsTrue(ipImage.IsValid, 'ipImage must contain an image');
Check.IsTrue(ipImage.HasChannelCount(1), 'ipImage must have 1 channel');

Check.IsTrue((eMorphType.Value = ETcVnMorphologicalOperator.TCVN_MO_OPENING) OR
             (eMorphType.Value = ETcVnMorphologicalOperator.TCVN_MO_CLOSING), 'eMorphType must be OPENING or CLOSING');

Check.IsTrue(nMinSize.IsOdd, 'nMinSize must be an odd number');
Check.IsTrue(nMinSize.Value >= 3, 'nMinSize must be greater than or equal to 3');

Check.IsTrue(nMaxSize.Value >= nMinSize.Value, 'nMaxSize must be greater than or equal to nMinSize');

Check.IsTrue(nStep.IsEven, 'nStep must be an even number');
Check.IsTrue(nStep.Value >= 2, 'nStep must be greater than or equal to 2');
END_METHOD

END_FUNCTION_BLOCK

// Nodes/Texture Analysis/Node_F_VN_HaralickFeatures
{attribute 'linkalways'} 
{attribute 'no_explicit_call' := 'This FB is a CLASS and must be accessed using methods or properties'}
{attribute 'enable_dynamic_creation'}
FUNCTION_BLOCK Node_F_VN_HaralickFeatures EXTENDS VisionNode
VAR
    ipImage : _ITcVnImage;
    ipFeatures : _ITcVnContainer;
    nDist : _UDINT(0);
    hrPrev : _HRESULT(S_OK);
	hresult : _HRESULT(S_OK);
END_VAR

METHOD FB_init : BOOL
VAR_INPUT
	bInitRetains : BOOL; // if TRUE, the retain variables are initialized (warm start / cold start)
	bInCopyCode : BOOL;  // if TRUE, the instance afterwards gets moved into the copy code (online change)
END_VAR
AddInput('ipImage', ipImage);
AddParameter('nDist', nDist);
AddInput('hrPrev', hrPrev);
AddOutput('ipFeatures', ipFeatures);
AddOutput('hresult',hresult);
END_METHOD

METHOD PUBLIC  Clone : I_Node
VAR
	pNode : POINTER TO Node_F_VN_HaralickFeatures;
END_VAR
pNode := __NEW(Node_F_VN_HaralickFeatures);
Clone := pNode^;
END_METHOD

METHOD PROTECTED OnExecute
hresult.Value := F_VN_HaralickFeatures(
    ipImage := ipImage.Value,
    ipFeatures := ipFeatures.Value,
    nDist := nDist.Value,
	hrPrev:= hrPrev.Value);
END_METHOD

METHOD PUBLIC PreExecutionCheck
VAR_INPUT
	Check : I_PreExecutionChecks;
END_VAR
Check.IsTrue(ipImage.IsValid, 'ipImage must contain an image');
Check.IsTrue(ipImage.HasChannelCount(1), 'ipImage must have 1 channel');
Check.IsTrue(ipImage.IsPixelDepth(8), 'ipImage must have 8 bit pixel depth');
END_METHOD

END_FUNCTION_BLOCK

// Nodes/VisionNode/VisionHardwareNode
FUNCTION_BLOCK ABSTRACT VisionHardwareNode EXTENDS HardwareNode IMPLEMENTS I_PreCheckedNode
VAR
	preExecutionCheckExtension : PreExecutionCheckExtension('precheck', THIS^);
END_VAR

METHOD PUBLIC Execute
IF NOT preExecutionCheckExtension.Check() THEN
	RETURN;
END_IF

SUPER^.Execute();
END_METHOD

METHOD PUBLIC ABSTRACT PreExecutionCheck
VAR_INPUT
	Check : I_PreExecutionChecks;
END_VAR
END_METHOD

END_FUNCTION_BLOCK

// Nodes/VisionNodePack
{attribute 'linkalways'} 
{attribute 'no_explicit_call' := 'This FB is a CLASS and must be accessed using methods or properties'}
{attribute 'enable_dynamic_creation'}
FUNCTION_BLOCK VisionNodePack
VAR
    // Algebraic Container Operations
    node_F_VN_AddToContainerElements_DINT : Node_F_VN_AddToContainerElements_DINT;
    node_F_VN_AddToContainerElements_INT : Node_F_VN_AddToContainerElements_INT;
    node_F_VN_AddToContainerElements_LREAL : Node_F_VN_AddToContainerElements_LREAL;
    node_F_VN_AddToContainerElements_REAL : Node_F_VN_AddToContainerElements_REAL;
    node_F_VN_AddToContainerElements_SINT : Node_F_VN_AddToContainerElements_SINT;
    node_F_VN_AddToContainerElements_TcVnKeyPoint : Node_F_VN_AddToContainerElements_TcVnKeyPoint;
    node_F_VN_AddToContainerElements_TcVnPoint2_DINT : Node_F_VN_AddToContainerElements_TcVnPoint2_DINT;
    node_F_VN_AddToContainerElements_TcVnPoint2_LREAL : Node_F_VN_AddToContainerElements_TcVnPoint2_LREAL;
    node_F_VN_AddToContainerElements_TcVnPoint2_REAL : Node_F_VN_AddToContainerElements_TcVnPoint2_REAL;
    node_F_VN_AddToContainerElements_TcVnPoint3_LREAL : Node_F_VN_AddToContainerElements_TcVnPoint3_LREAL;
    node_F_VN_AddToContainerElements_TcVnPoint3_REAL : Node_F_VN_AddToContainerElements_TcVnPoint3_REAL;
    node_F_VN_AddToContainerElements_TcVnRectangle_DINT : Node_F_VN_AddToContainerElements_TcVnRectangle_DINT;
    node_F_VN_AddToContainerElements_TcVnRotatedRectangle : Node_F_VN_AddToContainerElements_TcVnRotatedRectangle;
    node_F_VN_AddToContainerElements_TcVnVector2_DINT : Node_F_VN_AddToContainerElements_TcVnVector2_DINT;
    node_F_VN_AddToContainerElements_TcVnVector2_INT : Node_F_VN_AddToContainerElements_TcVnVector2_INT;
    node_F_VN_AddToContainerElements_TcVnVector2_REAL : Node_F_VN_AddToContainerElements_TcVnVector2_REAL;
    node_F_VN_AddToContainerElements_TcVnVector2_SINT : Node_F_VN_AddToContainerElements_TcVnVector2_SINT;
    node_F_VN_AddToContainerElements_TcVnVector2_UINT : Node_F_VN_AddToContainerElements_TcVnVector2_UINT;
    node_F_VN_AddToContainerElements_TcVnVector2_USINT : Node_F_VN_AddToContainerElements_TcVnVector2_USINT;
    node_F_VN_AddToContainerElements_TcVnVector3_INT : Node_F_VN_AddToContainerElements_TcVnVector3_INT;
    node_F_VN_AddToContainerElements_TcVnVector3_REAL : Node_F_VN_AddToContainerElements_TcVnVector3_REAL;
    node_F_VN_AddToContainerElements_TcVnVector3_SINT : Node_F_VN_AddToContainerElements_TcVnVector3_SINT;
    node_F_VN_AddToContainerElements_TcVnVector3_UINT : Node_F_VN_AddToContainerElements_TcVnVector3_UINT;
    node_F_VN_AddToContainerElements_TcVnVector3_USINT : Node_F_VN_AddToContainerElements_TcVnVector3_USINT;
    node_F_VN_AddToContainerElements_TcVnVector4_DINT : Node_F_VN_AddToContainerElements_TcVnVector4_DINT;
    node_F_VN_AddToContainerElements_TcVnVector4_INT : Node_F_VN_AddToContainerElements_TcVnVector4_INT;
    node_F_VN_AddToContainerElements_TcVnVector4_LREAL : Node_F_VN_AddToContainerElements_TcVnVector4_LREAL;
    node_F_VN_AddToContainerElements_TcVnVector4_REAL : Node_F_VN_AddToContainerElements_TcVnVector4_REAL;
    node_F_VN_AddToContainerElements_TcVnVector4_SINT : Node_F_VN_AddToContainerElements_TcVnVector4_SINT;
    node_F_VN_AddToContainerElements_TcVnVector4_UINT : Node_F_VN_AddToContainerElements_TcVnVector4_UINT;
    node_F_VN_AddToContainerElements_TcVnVector4_USINT : Node_F_VN_AddToContainerElements_TcVnVector4_USINT;
    node_F_VN_AddToContainerElements_UDINT : Node_F_VN_AddToContainerElements_UDINT;
    node_F_VN_AddToContainerElements_UINT : node_F_VN_AddToContainerElements_UINT;
    node_F_VN_AddToContainerElements_ULINT : Node_F_VN_AddToContainerElements_ULINT;
    node_F_VN_AddToContainerElements_USINT : Node_F_VN_AddToContainerElements_USINT;
    node_F_VN_AddContainers : Node_F_VN_AddContainers;
    node_F_VN_BitwiseAndContainers : Node_F_VN_BitwiseAndContainers;
    node_F_VN_BitwiseNotContainer : Node_F_VN_BitwiseNotContainer;
    node_F_VN_BitwiseOrContainers : Node_F_VN_BitwiseOrContainers;
    node_F_VN_BitwiseXorContainers : Node_F_VN_BitwiseXorContainers;
    node_F_VN_DivideContainers : Node_F_VN_DivideContainers;
    node_F_VN_DivideContainersExp : Node_F_VN_DivideContainersExp;
    node_F_VN_MaxContainer : Node_F_VN_MaxContainer;
    node_F_VN_MinContainer : Node_F_VN_MinContainer;
    node_F_VN_MultiplyContainers : Node_F_VN_MultiplyContainers;
    //node_F_VN_MultiplyWithContainerElements1 : Node_F_VN_MultiplyWithContainerElements1;
    //node_F_VN_MultiplyWithContainerElements1 : Node_F_VN_MultiplyWithContainerElements2;
    //node_F_VN_MultiplyWithContainerElements1 : Node_F_VN_MultiplyWithContainerElements3;
    //node_F_VN_MultiplyWithContainerElements1 : Node_F_VN_MultiplyWithContainerElements4;
    node_F_VN_NegateContainer : Node_F_VN_NegateContainer;
    node_F_VN_SubtractContainers : Node_F_VN_SubtractContainers;
   
    // Algebraic Image Operations
    node_F_VN_AddImages : Node_F_VN_AddImages;
    node_F_VN_AddImagesWeighted : Node_F_VN_AddImagesWeighted;
    node_F_VN_AddImagesWeightedExp : Node_F_VN_AddImagesWeightedExp;
    node_F_VN_AddScalarToImage : Node_F_VN_AddScalarToImage;
    node_F_VN_AddVectorToImage : Node_F_VN_AddVectorToImage;
    node_F_VN_BitwiseAndImages : Node_F_VN_BitwiseAndImages;
    node_F_VN_BitwiseAndImagesExp : Node_F_VN_BitwiseAndImagesExp;
    node_F_VN_BitwiseAndScalarWithImage : Node_F_VN_BitwiseAndScalarWithImage;
    node_F_VN_BitwiseAndVectorWithImage : Node_F_VN_BitwiseAndVectorWithImage;
    node_F_VN_BitwiseNotImage : Node_F_VN_BitwiseNotImage;
    node_F_VN_BitwiseNotImageExp : Node_F_VN_BitwiseNotImageExp;
    node_F_VN_BitwiseOrImages : Node_F_VN_BitwiseOrImages;
    node_F_VN_BitwiseOrImagesExp : Node_F_VN_BitwiseOrImagesExp;
    node_F_VN_BitwiseOrScalarWithImage : Node_F_VN_BitwiseOrScalarWithImage;
    node_F_VN_BitwiseOrVectorWithImage : Node_F_VN_BitwiseOrVectorWithImage;
    node_F_VN_BitwiseXorImages : Node_F_VN_BitwiseXorImages;
    node_F_VN_BitwiseXorImagesExp : Node_F_VN_BitwiseXorImagesExp;
    node_F_VN_BitwiseXorScalarWithImage : Node_F_VN_BitwiseXorScalarWithImage;
    node_F_VN_BitwiseXorVectorWithImage : Node_F_VN_BitwiseXorVectorWithImage;
    //node_F_VN_BlendImages : Node_F_VN_BlendImages;
    node_F_VN_DivideImageByScalar : Node_F_VN_DivideImageByScalar;
    node_F_VN_DivideImageByVector : Node_F_VN_DivideImageByVector;
    node_F_VN_DivideImages : Node_F_VN_DivideImages;
    node_F_VN_DivideScalarByImage : Node_F_VN_DivideScalarByImage;
    node_F_VN_DivideVectorByImage : Node_F_VN_DivideVectorByImage;
    node_F_VN_ElementwiseExp : Node_F_VN_ElementwiseExp;
    node_F_VN_ElementwiseLog : Node_F_VN_ElementwiseLog;
    node_F_VN_MaxImage : Node_F_VN_MaxImage;
    node_F_VN_MaxImageExp : Node_F_VN_MaxImageExp;
    node_F_VN_MaxImageWithScalar : Node_F_VN_MaxImageWithScalar;
    node_F_VN_MaxImageWithScalarExp : Node_F_VN_MaxImageWithScalarExp;
    node_F_VN_MaxImageWithVector : Node_F_VN_MaxImageWithVector;
    node_F_VN_MaxImageWithVectorExp : Node_F_VN_MaxImageWithVectorExp;
    node_F_VN_MinImage : Node_F_VN_MinImage;
    node_F_VN_MinImageExp : Node_F_VN_MinImageExp;
    node_F_VN_MinImageWithScalar : Node_F_VN_MinImageWithScalar;
    node_F_VN_MinImageWithScalarExp : Node_F_VN_MinImageWithScalarExp;
    node_F_VN_MinImageWithVector : Node_F_VN_MinImageWithVector;
    node_F_VN_MinImageWithVectorExp : Node_F_VN_MinImageWithVectorExp;
    node_F_VN_MultiplyImages : Node_F_VN_MultiplyImages;
    node_F_VN_MultiplyImageWithScalar : Node_F_VN_MultiplyImageWithScalar;
    node_F_VN_MultiplyImageWithVector : Node_F_VN_MultiplyImageWithVector;
    node_F_VN_SubtractImageFromScalar : Node_F_VN_SubtractImageFromScalar;
    node_F_VN_SubtractImageFromVector : Node_F_VN_SubtractImageFromVector;
    node_F_VN_SubtractImages : Node_F_VN_SubtractImages;
    node_F_VN_SubtractScalarFromImage : Node_F_VN_SubtractScalarFromImage;
    node_F_VN_SubtractVectorFromImage : Node_F_VN_SubtractVectorFromImage;
        
    // Basic Container Operations
    node_F_VN_AppendToContainer_DINT : Node_F_VN_AppendToContainer_DINT;
    node_F_VN_AppendToContainer_INT : Node_F_VN_AppendToContainer_INT;
    node_F_VN_AppendToContainer_ITcVnContainer : Node_F_VN_AppendToContainer_ITcVnContainer;
    //node_F_VN_AppendToContainer_ITcVnForwardIterator : Node_F_VN_AppendToContainer_ITcVnForwardIterator;
    node_F_VN_AppendToContainer_ITcVnImage : Node_F_VN_AppendToContainer_ITcVnImage;
    node_F_VN_AppendToContainer_LREAL : Node_F_VN_AppendToContainer_LREAL;
    node_F_VN_AppendToContainer_REAL : Node_F_VN_AppendToContainer_REAL;
    node_F_VN_AppendToContainer_SINT : Node_F_VN_AppendToContainer_SINT;
    node_F_VN_AppendToContainer_TcVnDMatch : Node_F_VN_AppendToContainer_TcVnDMatch;
    node_F_VN_AppendToContainer_TcVnKeyPoint : Node_F_VN_AppendToContainer_TcVnKeyPoint;
    node_F_VN_AppendToContainer_TcVnPoint2_DINT : Node_F_VN_AppendToContainer_TcVnPoint2_DINT;
    node_F_VN_AppendToContainer_TcVnPoint2_LREAL : Node_F_VN_AppendToContainer_TcVnPoint2_LREAL;
    node_F_VN_AppendToContainer_TcVnPoint2_REAL : Node_F_VN_AppendToContainer_TcVnPoint2_REAL;
    node_F_VN_AppendToContainer_TcVnPoint3_LREAL : Node_F_VN_AppendToContainer_TcVnPoint3_LREAL;
    node_F_VN_AppendToContainer_TcVnPoint3_REAL : Node_F_VN_AppendToContainer_TcVnPoint3_REAL;
    node_F_VN_AppendToContainer_TcVnRectangle_DINT : Node_F_VN_AppendToContainer_TcVnRectangle_DINT;
    node_F_VN_AppendToContainer_TcVnRotatedRectangle : Node_F_VN_AppendToContainer_TcVnRotatedRectangle;
    node_F_VN_AppendToContainer_TcVnVector2_DINT : Node_F_VN_AppendToContainer_TcVnVector2_DINT;
    node_F_VN_AppendToContainer_TcVnVector2_INT : Node_F_VN_AppendToContainer_TcVnVector2_INT;
    node_F_VN_AppendToContainer_TcVnVector2_REAL : Node_F_VN_AppendToContainer_TcVnVector2_REAL;
    node_F_VN_AppendToContainer_TcVnVector2_SINT : Node_F_VN_AppendToContainer_TcVnVector2_SINT;
    node_F_VN_AppendToContainer_TcVnVector2_UINT : Node_F_VN_AppendToContainer_TcVnVector2_UINT;
    node_F_VN_AppendToContainer_TcVnVector2_USINT : Node_F_VN_AppendToContainer_TcVnVector2_USINT;
    node_F_VN_AppendToContainer_TcVnVector3_INT : Node_F_VN_AppendToContainer_TcVnVector3_INT;
    node_F_VN_AppendToContainer_TcVnVector3_REAL : Node_F_VN_AppendToContainer_TcVnVector3_REAL;
    node_F_VN_AppendToContainer_TcVnVector3_SINT : Node_F_VN_AppendToContainer_TcVnVector3_SINT;
    node_F_VN_AppendToContainer_TcVnVector3_UINT : Node_F_VN_AppendToContainer_TcVnVector3_UINT;
    node_F_VN_AppendToContainer_TcVnVector3_USINT : Node_F_VN_AppendToContainer_TcVnVector3_USINT;
    node_F_VN_AppendToContainer_TcVnVector4_DINT : Node_F_VN_AppendToContainer_TcVnVector4_DINT;
    node_F_VN_AppendToContainer_TcVnVector4_INT : Node_F_VN_AppendToContainer_TcVnVector4_INT;
    node_F_VN_AppendToContainer_TcVnVector4_LREAL : Node_F_VN_AppendToContainer_TcVnVector4_LREAL;
    node_F_VN_AppendToContainer_TcVnVector4_REAL : Node_F_VN_AppendToContainer_TcVnVector4_REAL;
    node_F_VN_AppendToContainer_TcVnVector4_SINT : Node_F_VN_AppendToContainer_TcVnVector4_SINT;
    node_F_VN_AppendToContainer_TcVnVector4_UINT : Node_F_VN_AppendToContainer_TcVnVector4_UINT;
    node_F_VN_AppendToContainer_TcVnVector4_USINT : Node_F_VN_AppendToContainer_TcVnVector4_USINT;
    node_F_VN_AppendToContainer_UDINT : Node_F_VN_AppendToContainer_UDINT;
    node_F_VN_AppendToContainer_UINT : node_F_VN_AppendToContainer_UINT;
    node_F_VN_AppendToContainer_ULINT : Node_F_VN_AppendToContainer_ULINT;
    node_F_VN_AppendToContainer_USINT : Node_F_VN_AppendToContainer_USINT;
    
    node_F_VN_FillContainer_DINT : Node_F_VN_FillContainer_DINT;
    node_F_VN_FillContainer_INT : Node_F_VN_FillContainer_INT;
    node_F_VN_FillContainer_ITcVnImage : Node_F_VN_FillContainer_ITcVnImage;
    node_F_VN_FillContainer_LREAL : Node_F_VN_FillContainer_LREAL;
    node_F_VN_FillContainer_REAL : Node_F_VN_FillContainer_REAL;
    node_F_VN_FillContainer_SINT : Node_F_VN_FillContainer_SINT;
    node_F_VN_FillContainer_TcVnDMatch : Node_F_VN_FillContainer_TcVnDMatch;
    node_F_VN_FillContainer_TcVnKeyPoint : Node_F_VN_FillContainer_TcVnKeyPoint;
    node_F_VN_FillContainer_TcVnPoint2_DINT : Node_F_VN_FillContainer_TcVnPoint2_DINT;
    node_F_VN_FillContainer_TcVnPoint2_LREAL : Node_F_VN_FillContainer_TcVnPoint2_LREAL;
    node_F_VN_FillContainer_TcVnPoint2_REAL : Node_F_VN_FillContainer_TcVnPoint2_REAL;
    node_F_VN_FillContainer_TcVnPoint3_LREAL : Node_F_VN_FillContainer_TcVnPoint3_LREAL;
    node_F_VN_FillContainer_TcVnPoint3_REAL : Node_F_VN_FillContainer_TcVnPoint3_REAL;
    node_F_VN_FillContainer_TcVnRectangle_DINT : Node_F_VN_FillContainer_TcVnRectangle_DINT;
    node_F_VN_FillContainer_TcVnRotatedRectangle : Node_F_VN_FillContainer_TcVnRotatedRectangle;
    node_F_VN_FillContainer_TcVnVector2_DINT : Node_F_VN_FillContainer_TcVnVector2_DINT;
    node_F_VN_FillContainer_TcVnVector2_INT : Node_F_VN_FillContainer_TcVnVector2_INT;
    node_F_VN_FillContainer_TcVnVector2_REAL : Node_F_VN_FillContainer_TcVnVector2_REAL;
    node_F_VN_FillContainer_TcVnVector2_SINT : Node_F_VN_FillContainer_TcVnVector2_SINT;
    node_F_VN_FillContainer_TcVnVector2_UINT : Node_F_VN_FillContainer_TcVnVector2_UINT;
    node_F_VN_FillContainer_TcVnVector2_USINT : Node_F_VN_FillContainer_TcVnVector2_USINT;
    node_F_VN_FillContainer_TcVnVector3_INT : Node_F_VN_FillContainer_TcVnVector3_INT;
    node_F_VN_FillContainer_TcVnVector3_REAL : Node_F_VN_FillContainer_TcVnVector3_REAL;
    node_F_VN_FillContainer_TcVnVector3_SINT : Node_F_VN_FillContainer_TcVnVector3_SINT;
    node_F_VN_FillContainer_TcVnVector3_UINT : Node_F_VN_FillContainer_TcVnVector3_UINT;
    node_F_VN_FillContainer_TcVnVector3_USINT : Node_F_VN_FillContainer_TcVnVector3_USINT;
    node_F_VN_FillContainer_TcVnVector4_DINT : Node_F_VN_FillContainer_TcVnVector4_DINT;
    node_F_VN_FillContainer_TcVnVector4_INT : Node_F_VN_FillContainer_TcVnVector4_INT;
    node_F_VN_FillContainer_TcVnVector4_LREAL : Node_F_VN_FillContainer_TcVnVector4_LREAL;
    node_F_VN_FillContainer_TcVnVector4_REAL : Node_F_VN_FillContainer_TcVnVector4_REAL;
    node_F_VN_FillContainer_TcVnVector4_SINT : Node_F_VN_FillContainer_TcVnVector4_SINT;
    node_F_VN_FillContainer_TcVnVector4_UINT : Node_F_VN_FillContainer_TcVnVector4_UINT;
    node_F_VN_FillContainer_TcVnVector4_USINT : Node_F_VN_FillContainer_TcVnVector4_USINT;
    node_F_VN_FillContainer_UDINT : Node_F_VN_FillContainer_UDINT;
    node_F_VN_FillContainer_UINT : node_F_VN_FillContainer_UINT;
    node_F_VN_FillContainer_ULINT : Node_F_VN_FillContainer_ULINT;
    node_F_VN_FillContainer_USINT : Node_F_VN_FillContainer_USINT;
    
    node_F_VN_FillContainerExp_DINT : Node_F_VN_FillContainerExp_DINT;
    node_F_VN_FillContainerExp_INT : Node_F_VN_FillContainerExp_INT;
    node_F_VN_FillContainerExp_ITcVnImage : Node_F_VN_FillContainerExp_ITcVnImage;
    node_F_VN_FillContainerExp_LREAL : Node_F_VN_FillContainerExp_LREAL;
    node_F_VN_FillContainerExp_REAL : Node_F_VN_FillContainerExp_REAL;
    node_F_VN_FillContainerExp_SINT : Node_F_VN_FillContainerExp_SINT;
    node_F_VN_FillContainerExp_TcVnDMatch : Node_F_VN_FillContainerExp_TcVnDMatch;
    node_F_VN_FillContainerExp_TcVnKeyPoint : Node_F_VN_FillContainerExp_TcVnKeyPoint;
    node_F_VN_FillContainerExp_TcVnPoint2_DINT : Node_F_VN_FillContainerExp_TcVnPoint2_DINT;
    node_F_VN_FillContainerExp_TcVnPoint2_LREAL : Node_F_VN_FillContainerExp_TcVnPoint2_LREAL;
    node_F_VN_FillContainerExp_TcVnPoint2_REAL : Node_F_VN_FillContainerExp_TcVnPoint2_REAL;
    node_F_VN_FillContainerExp_TcVnPoint3_LREAL : Node_F_VN_FillContainerExp_TcVnPoint3_LREAL;
    node_F_VN_FillContainerExp_TcVnPoint3_REAL : Node_F_VN_FillContainerExp_TcVnPoint3_REAL;
    node_F_VN_FillContainerExp_TcVnRectangle_DINT : Node_F_VN_FillContainerExp_TcVnRectangle_DINT;
    node_F_VN_FillContainerExp_TcVnRotatedRectangle : Node_F_VN_FillContainerExp_TcVnRotatedRectangle;
    node_F_VN_FillContainerExp_TcVnVector2_DINT : Node_F_VN_FillContainerExp_TcVnVector2_DINT;
    node_F_VN_FillContainerExp_TcVnVector2_INT : Node_F_VN_FillContainerExp_TcVnVector2_INT;
    node_F_VN_FillContainerExp_TcVnVector2_REAL : Node_F_VN_FillContainerExp_TcVnVector2_REAL;
    node_F_VN_FillContainerExp_TcVnVector2_SINT : Node_F_VN_FillContainerExp_TcVnVector2_SINT;
    node_F_VN_FillContainerExp_TcVnVector2_UINT : Node_F_VN_FillContainerExp_TcVnVector2_UINT;
    node_F_VN_FillContainerExp_TcVnVector2_USINT : Node_F_VN_FillContainerExp_TcVnVector2_USINT;
    node_F_VN_FillContainerExp_TcVnVector3_INT : Node_F_VN_FillContainerExp_TcVnVector3_INT;
    node_F_VN_FillContainerExp_TcVnVector3_REAL : Node_F_VN_FillContainerExp_TcVnVector3_REAL;
    node_F_VN_FillContainerExp_TcVnVector3_SINT : Node_F_VN_FillContainerExp_TcVnVector3_SINT;
    node_F_VN_FillContainerExp_TcVnVector3_UINT : Node_F_VN_FillContainerExp_TcVnVector3_UINT;
    node_F_VN_FillContainerExp_TcVnVector3_USINT : Node_F_VN_FillContainerExp_TcVnVector3_USINT;
    node_F_VN_FillContainerExp_TcVnVector4_DINT : Node_F_VN_FillContainerExp_TcVnVector4_DINT;
    node_F_VN_FillContainerExp_TcVnVector4_INT : Node_F_VN_FillContainerExp_TcVnVector4_INT;
    node_F_VN_FillContainerExp_TcVnVector4_LREAL : Node_F_VN_FillContainerExp_TcVnVector4_LREAL;
    node_F_VN_FillContainerExp_TcVnVector4_REAL : Node_F_VN_FillContainerExp_TcVnVector4_REAL;
    node_F_VN_FillContainerExp_TcVnVector4_SINT : Node_F_VN_FillContainerExp_TcVnVector4_SINT;
    node_F_VN_FillContainerExp_TcVnVector4_UINT : Node_F_VN_FillContainerExp_TcVnVector4_UINT;
    node_F_VN_FillContainerExp_TcVnVector4_USINT : Node_F_VN_FillContainerExp_TcVnVector4_USINT;
    node_F_VN_FillContainerExp_UDINT : Node_F_VN_FillContainerExp_UDINT;
    node_F_VN_FillContainerExp_UINT : node_F_VN_FillContainerExp_UINT;
    node_F_VN_FillContainerExp_ULINT : Node_F_VN_FillContainerExp_ULINT;
    node_F_VN_FillContainerExp_USINT : Node_F_VN_FillContainerExp_USINT;
    
    node_F_VN_GetAt_DINT : Node_F_VN_GetAt_DINT;
    node_F_VN_GetAt_INT : Node_F_VN_GetAt_INT;
    node_F_VN_GetAt_ITcVnContainer : Node_F_VN_GetAt_ITcVnContainer;
    node_F_VN_GetAt_ITcVnImage : Node_F_VN_GetAt_ITcVnImage;
    node_F_VN_GetAt_LREAL : Node_F_VN_GetAt_LREAL;
    node_F_VN_GetAt_REAL : Node_F_VN_GetAt_REAL;
    node_F_VN_GetAt_SINT : Node_F_VN_GetAt_SINT;
    node_F_VN_GetAt_TcVnDMatch : Node_F_VN_GetAt_TcVnDMatch;
    node_F_VN_GetAt_TcVnKeyPoint : Node_F_VN_GetAt_TcVnKeyPoint;
    node_F_VN_GetAt_TcVnPoint2_DINT : Node_F_VN_GetAt_TcVnPoint2_DINT;
    node_F_VN_GetAt_TcVnPoint2_LREAL : Node_F_VN_GetAt_TcVnPoint2_LREAL;
    node_F_VN_GetAt_TcVnPoint2_REAL : Node_F_VN_GetAt_TcVnPoint2_REAL;
    node_F_VN_GetAt_TcVnPoint3_LREAL : Node_F_VN_GetAt_TcVnPoint3_LREAL;
    node_F_VN_GetAt_TcVnPoint3_REAL : Node_F_VN_GetAt_TcVnPoint3_REAL;
    node_F_VN_GetAt_TcVnRectangle_DINT : Node_F_VN_GetAt_TcVnRectangle_DINT;
    node_F_VN_GetAt_TcVnRotatedRectangle : Node_F_VN_GetAt_TcVnRotatedRectangle;
    node_F_VN_GetAt_TcVnVector2_DINT : Node_F_VN_GetAt_TcVnVector2_DINT;
    node_F_VN_GetAt_TcVnVector2_INT : Node_F_VN_GetAt_TcVnVector2_INT;
    node_F_VN_GetAt_TcVnVector2_REAL : Node_F_VN_GetAt_TcVnVector2_REAL;
    node_F_VN_GetAt_TcVnVector2_SINT : Node_F_VN_GetAt_TcVnVector2_SINT;
    node_F_VN_GetAt_TcVnVector2_UINT : Node_F_VN_GetAt_TcVnVector2_UINT;
    node_F_VN_GetAt_TcVnVector2_USINT : Node_F_VN_GetAt_TcVnVector2_USINT;
    node_F_VN_GetAt_TcVnVector3_INT : Node_F_VN_GetAt_TcVnVector3_INT;
    node_F_VN_GetAt_TcVnVector3_REAL : Node_F_VN_GetAt_TcVnVector3_REAL;
    node_F_VN_GetAt_TcVnVector3_SINT : Node_F_VN_GetAt_TcVnVector3_SINT;
    node_F_VN_GetAt_TcVnVector3_UINT : Node_F_VN_GetAt_TcVnVector3_UINT;
    node_F_VN_GetAt_TcVnVector3_USINT : Node_F_VN_GetAt_TcVnVector3_USINT;
    node_F_VN_GetAt_TcVnVector4_DINT : Node_F_VN_GetAt_TcVnVector4_DINT;
    node_F_VN_GetAt_TcVnVector4_INT : Node_F_VN_GetAt_TcVnVector4_INT;
    node_F_VN_GetAt_TcVnVector4_LREAL : Node_F_VN_GetAt_TcVnVector4_LREAL;
    node_F_VN_GetAt_TcVnVector4_REAL : Node_F_VN_GetAt_TcVnVector4_REAL;
    node_F_VN_GetAt_TcVnVector4_SINT : Node_F_VN_GetAt_TcVnVector4_SINT;
    node_F_VN_GetAt_TcVnVector4_UINT : Node_F_VN_GetAt_TcVnVector4_UINT;
    node_F_VN_GetAt_TcVnVector4_USINT : Node_F_VN_GetAt_TcVnVector4_USINT;
    node_F_VN_GetAt_UDINT : Node_F_VN_GetAt_UDINT;
    node_F_VN_GetAt_UINT : node_F_VN_GetAt_UINT;
    node_F_VN_GetAt_ULINT : Node_F_VN_GetAt_ULINT;
    node_F_VN_GetAt_USINT : Node_F_VN_GetAt_USINT;
    
    node_F_VN_InsertIntoContainer_DINT : Node_F_VN_InsertIntoContainer_DINT;
    node_F_VN_InsertIntoContainer_INT : Node_F_VN_InsertIntoContainer_INT;
    node_F_VN_InsertIntoContainer_ITcVnContainer : Node_F_VN_InsertIntoContainer_ITcVnContainer;
    //node_F_VN_InsertIntoContainer_ITcVnForwardIterator : Node_F_VN_InsertIntoContainer_ITcVnForwardIterator;
    node_F_VN_InsertIntoContainer_ITcVnImage : Node_F_VN_InsertIntoContainer_ITcVnImage;
    node_F_VN_InsertIntoContainer_LREAL : Node_F_VN_InsertIntoContainer_LREAL;
    node_F_VN_InsertIntoContainer_REAL : Node_F_VN_InsertIntoContainer_REAL;
    node_F_VN_InsertIntoContainer_SINT : Node_F_VN_InsertIntoContainer_SINT;
    node_F_VN_InsertIntoContainer_TcVnDMatch : Node_F_VN_InsertIntoContainer_TcVnDMatch;
    node_F_VN_InsertIntoContainer_TcVnKeyPoint : Node_F_VN_InsertIntoContainer_TcVnKeyPoint;
    node_F_VN_InsertIntoContainer_TcVnPoint2_DINT : Node_F_VN_InsertIntoContainer_TcVnPoint2_DINT;
    node_F_VN_InsertIntoContainer_TcVnPoint2_LREAL : Node_F_VN_InsertIntoContainer_TcVnPoint2_LREAL;
    node_F_VN_InsertIntoContainer_TcVnPoint2_REAL : Node_F_VN_InsertIntoContainer_TcVnPoint2_REAL;
    node_F_VN_InsertIntoContainer_TcVnPoint3_LREAL : Node_F_VN_InsertIntoContainer_TcVnPoint3_LREAL;
    node_F_VN_InsertIntoContainer_TcVnPoint3_REAL : Node_F_VN_InsertIntoContainer_TcVnPoint3_REAL;
    node_F_VN_InsertIntoContainer_TcVnRectangle_DINT : Node_F_VN_InsertIntoContainer_TcVnRectangle_DINT;
    node_F_VN_InsertIntoContainer_TcVnRotatedRectangle : Node_F_VN_InsertIntoContainer_TcVnRotatedRectangle;
    node_F_VN_InsertIntoContainer_TcVnVector2_DINT : Node_F_VN_InsertIntoContainer_TcVnVector2_DINT;
    node_F_VN_InsertIntoContainer_TcVnVector2_INT : Node_F_VN_InsertIntoContainer_TcVnVector2_INT;
    node_F_VN_InsertIntoContainer_TcVnVector2_REAL : Node_F_VN_InsertIntoContainer_TcVnVector2_REAL;
    node_F_VN_InsertIntoContainer_TcVnVector2_SINT : Node_F_VN_InsertIntoContainer_TcVnVector2_SINT;
    node_F_VN_InsertIntoContainer_TcVnVector2_UINT : Node_F_VN_InsertIntoContainer_TcVnVector2_UINT;
    node_F_VN_InsertIntoContainer_TcVnVector2_USINT : Node_F_VN_InsertIntoContainer_TcVnVector2_USINT;
    node_F_VN_InsertIntoContainer_TcVnVector3_INT : Node_F_VN_InsertIntoContainer_TcVnVector3_INT;
    node_F_VN_InsertIntoContainer_TcVnVector3_REAL : Node_F_VN_InsertIntoContainer_TcVnVector3_REAL;
    node_F_VN_InsertIntoContainer_TcVnVector3_SINT : Node_F_VN_InsertIntoContainer_TcVnVector3_SINT;
    node_F_VN_InsertIntoContainer_TcVnVector3_UINT : Node_F_VN_InsertIntoContainer_TcVnVector3_UINT;
    node_F_VN_InsertIntoContainer_TcVnVector3_USINT : Node_F_VN_InsertIntoContainer_TcVnVector3_USINT;
    node_F_VN_InsertIntoContainer_TcVnVector4_DINT : Node_F_VN_InsertIntoContainer_TcVnVector4_DINT;
    node_F_VN_InsertIntoContainer_TcVnVector4_INT : Node_F_VN_InsertIntoContainer_TcVnVector4_INT;
    node_F_VN_InsertIntoContainer_TcVnVector4_LREAL : Node_F_VN_InsertIntoContainer_TcVnVector4_LREAL;
    node_F_VN_InsertIntoContainer_TcVnVector4_REAL : Node_F_VN_InsertIntoContainer_TcVnVector4_REAL;
    node_F_VN_InsertIntoContainer_TcVnVector4_SINT : Node_F_VN_InsertIntoContainer_TcVnVector4_SINT;
    node_F_VN_InsertIntoContainer_TcVnVector4_UINT : Node_F_VN_InsertIntoContainer_TcVnVector4_UINT;
    node_F_VN_InsertIntoContainer_TcVnVector4_USINT : Node_F_VN_InsertIntoContainer_TcVnVector4_USINT;
    node_F_VN_InsertIntoContainer_UDINT : Node_F_VN_InsertIntoContainer_UDINT;
    node_F_VN_InsertIntoContainer_UINT : node_F_VN_InsertIntoContainer_UINT;
    node_F_VN_InsertIntoContainer_ULINT : Node_F_VN_InsertIntoContainer_ULINT;
    node_F_VN_InsertIntoContainer_USINT : Node_F_VN_InsertIntoContainer_USINT;
    
    node_F_VN_SetAt_DINT : Node_F_VN_SetAt_DINT;
    node_F_VN_SetAt_INT : Node_F_VN_SetAt_INT;
    node_F_VN_SetAt_ITcVnContainer : Node_F_VN_SetAt_ITcVnContainer;
    node_F_VN_SetAt_ITcVnImage : Node_F_VN_SetAt_ITcVnImage;
    node_F_VN_SetAt_LREAL : Node_F_VN_SetAt_LREAL;
    node_F_VN_SetAt_REAL : Node_F_VN_SetAt_REAL;
    node_F_VN_SetAt_SINT : Node_F_VN_SetAt_SINT;
    node_F_VN_SetAt_TcVnDMatch : Node_F_VN_SetAt_TcVnDMatch;
    node_F_VN_SetAt_TcVnKeyPoint : Node_F_VN_SetAt_TcVnKeyPoint;
    node_F_VN_SetAt_TcVnPoint2_DINT : Node_F_VN_SetAt_TcVnPoint2_DINT;
    node_F_VN_SetAt_TcVnPoint2_LREAL : Node_F_VN_SetAt_TcVnPoint2_LREAL;
    node_F_VN_SetAt_TcVnPoint2_REAL : Node_F_VN_SetAt_TcVnPoint2_REAL;
    node_F_VN_SetAt_TcVnPoint3_LREAL : Node_F_VN_SetAt_TcVnPoint3_LREAL;
    node_F_VN_SetAt_TcVnPoint3_REAL : Node_F_VN_SetAt_TcVnPoint3_REAL;
    node_F_VN_SetAt_TcVnRectangle_DINT : Node_F_VN_SetAt_TcVnRectangle_DINT;
    node_F_VN_SetAt_TcVnRotatedRectangle : Node_F_VN_SetAt_TcVnRotatedRectangle;
    node_F_VN_SetAt_TcVnVector2_DINT : Node_F_VN_SetAt_TcVnVector2_DINT;
    node_F_VN_SetAt_TcVnVector2_INT : Node_F_VN_SetAt_TcVnVector2_INT;
    node_F_VN_SetAt_TcVnVector2_REAL : Node_F_VN_SetAt_TcVnVector2_REAL;
    node_F_VN_SetAt_TcVnVector2_SINT : Node_F_VN_SetAt_TcVnVector2_SINT;
    node_F_VN_SetAt_TcVnVector2_UINT : Node_F_VN_SetAt_TcVnVector2_UINT;
    node_F_VN_SetAt_TcVnVector2_USINT : Node_F_VN_SetAt_TcVnVector2_USINT;
    node_F_VN_SetAt_TcVnVector3_INT : Node_F_VN_SetAt_TcVnVector3_INT;
    node_F_VN_SetAt_TcVnVector3_REAL : Node_F_VN_SetAt_TcVnVector3_REAL;
    node_F_VN_SetAt_TcVnVector3_SINT : Node_F_VN_SetAt_TcVnVector3_SINT;
    node_F_VN_SetAt_TcVnVector3_UINT : Node_F_VN_SetAt_TcVnVector3_UINT;
    node_F_VN_SetAt_TcVnVector3_USINT : Node_F_VN_SetAt_TcVnVector3_USINT;
    node_F_VN_SetAt_TcVnVector4_DINT : Node_F_VN_SetAt_TcVnVector4_DINT;
    node_F_VN_SetAt_TcVnVector4_INT : Node_F_VN_SetAt_TcVnVector4_INT;
    node_F_VN_SetAt_TcVnVector4_LREAL : Node_F_VN_SetAt_TcVnVector4_LREAL;
    node_F_VN_SetAt_TcVnVector4_REAL : Node_F_VN_SetAt_TcVnVector4_REAL;
    node_F_VN_SetAt_TcVnVector4_SINT : Node_F_VN_SetAt_TcVnVector4_SINT;
    node_F_VN_SetAt_TcVnVector4_UINT : Node_F_VN_SetAt_TcVnVector4_UINT;
    node_F_VN_SetAt_TcVnVector4_USINT : Node_F_VN_SetAt_TcVnVector4_USINT;
    node_F_VN_SetAt_UDINT : Node_F_VN_SetAt_UDINT;
    node_F_VN_SetAt_UINT : node_F_VN_SetAt_UINT;
    node_F_VN_SetAt_ULINT : Node_F_VN_SetAt_ULINT;
    node_F_VN_SetAt_USINT : Node_F_VN_SetAt_USINT;
    
    //node_F_VN_AdvanceIterator : Node_F_VN_AdvanceIterator;
    node_F_VN_CheckIfEmpty : Node_F_VN_CheckIfEmpty;
    //node_F_VN_CheckIfIteratorIsAtEnd : Node_F_VN_CheckIfIteratorIsAtEnd;
    //node_F_VN_ConvertContainerType : Node_F_VN_ConvertContainerType;
    node_F_VN_CopyContainer : Node_F_VN_CopyContainer;
    //node_F_VN_CopyContainerElementsConditional_ITcVnContainer : Node_F_VN_CopyContainerElementsConditional_ITcVnContainer;
    //node_F_VN_CopyContainerElementsConditional_ITcVnForwardIterator : Node_F_VN_CopyContainerElementsConditional_ITcVnForwardIterator;
	node_F_VN_CreateContainer : Node_F_VN_CreateContainer;
    //node_F_VN_CreateContainerFromArray : Node_F_VN_CreateContainerFromArray;
    //node_F_VN_EraseFromContainer : Node_F_VN_EraseFromContainer;
    //node_F_VN_ExportContainer : Node_F_VN_ExportContainer;
    node_F_VN_ExportContainer_String : Node_F_VN_ExportContainer_String;
    //node_F_VN_ExportContainerSize : Node_F_VN_ExportContainerSize;
    //node_F_VN_ExportSubContainer : Node_F_VN_ExportSubContainer;
    node_F_VN_ExportSubContainer_String : Node_F_VN_ExportSubContainer_String;
    //node_F_VN_ExportSubContainerSize : Node_F_VN_ExportSubContainerSize;
    //node_F_VN_ExtractContainerRange : Node_F_VN_ExtractContainerRange;
    node_F_VN_ExtractContainerRange : Node_F_VN_ExtractContainerRange;
    //node_F_VN_GetContainer : Node_F_VN_GetContainer;
    //node_F_VN_GetContainerExp : Node_F_VN_GetContainerExp;
    //node_F_VN_GetForwardIterator : Node_F_VN_GetForwardIterator;
    node_F_VN_GetNumberOfElements : Node_F_VN_GetNumberOfElements;
    //node_F_VN_GetRandomAccessIterator : Node_F_VN_GetRandomAccessIterator;
    //node_F_VN_IncrementIterator : Node_F_VN_IncrementIterator;
    //node_F_VN_IteratorDistance : Node_F_VN_IteratorDistance;
    //node_F_VN_ReserveContainerMemory : Node_F_VN_ReserveContainerMemory;
    node_F_VN_ReverseContainer : Node_F_VN_ReverseContainer;
    //node_F_VN_SetContainer : Node_F_VN_SetContainer;
    //node_F_VN_SetIteratorToBegin : Node_F_VN_SetIteratorToBegin;
    
    // Basic Image Operations
    //node_F_VN_CombineImageChannels : Node_F_VN_CombineImageChannels;
    node_F_VN_ConvertElementType : Node_F_VN_ConvertElementType;
    node_F_VN_ConvertElementTypeExp : Node_F_VN_ConvertElementTypeExp;
    node_F_VN_CopyImage : Node_F_VN_CopyImage;
    node_F_VN_CopyImageRegion : Node_F_VN_CopyImageRegion;
    node_F_VN_CopyImageRegionToRegion : Node_F_VN_CopyImageRegionToRegion;
    node_F_VN_CopyIntoDisplayableImage : Node_F_VN_CopyIntoDisplayableImage;
    node_F_VN_CreateAssociatedImage : Node_F_VN_CreateAssociatedImage;
    node_F_VN_CreateEmptyImage : Node_F_VN_CreateEmptyImage;
    node_F_VN_CreateImage : Node_F_VN_CreateImage;
    node_F_VN_CreateImageAndSetPixels : Node_F_VN_CreateImageAndSetPixels;
    //node_F_VN_CreateImageFromArray : Node_F_VN_CreateImageFromArray;
    //node_F_VN_ExportImage : Node_F_VN_ExportImage;
    //node_F_VN_ExportImageAsBmp : Node_F_VN_ExportImageAsBmp;
    //node_F_VN_ExportImageAsBmpExp : Node_F_VN_ExportImageAsBmpExp;
    node_F_VN_ExportImageAsBmpSize : Node_F_VN_ExportImageAsBmpSize;
    node_F_VN_ExportImageAsBmpSizeExp : Node_F_VN_ExportImageAsBmpSizeExp;
    node_F_VN_ExportImageSize : Node_F_VN_ExportImageSize;
    node_F_VN_FuseImages : Node_F_VN_FuseImages;
    //node_F_VN_FuseImagesArray : Node_F_VN_FuseImagesArray;
    node_F_VN_GetImageChannel : Node_F_VN_GetImageChannel;
    node_F_VN_GetImageHeight : Node_F_VN_GetImageHeight;
    node_F_VN_GetImageInfo : Node_F_VN_GetImageInfo;
    node_F_VN_GetImageWidth : Node_F_VN_GetImageWidth;
    node_F_VN_GetPixel : Node_F_VN_GetPixel;
    node_F_VN_GetPixelFormat : Node_F_VN_GetPixelFormat;
    node_F_VN_GetRoi : Node_F_VN_GetRoi;
    node_F_VN_MixImageChannels : Node_F_VN_MixImageChannels;
    node_F_VN_ResetRoi : Node_F_VN_ResetRoi;
    node_F_VN_SetImageChannel : Node_F_VN_SetImageChannel;
    node_F_VN_SetPixel : Node_F_VN_SetPixel;
    node_F_VN_SetPixels : Node_F_VN_SetPixels;
    node_F_VN_SetPixelsExp : Node_F_VN_SetPixelsExp;
    node_F_VN_SetRoi : Node_F_VN_SetRoi;
    node_F_VN_SetRoi_TcVnRectangle_DINT : Node_F_VN_SetRoi_TcVnRectangle_DINT;
    node_F_VN_SetRoi_TcVnRectangle_UDINT : Node_F_VN_SetRoi_TcVnRectangle_UDINT;
    //node_F_VN_SplitImageChannels : Node_F_VN_SplitImageChannels;
    node_F_VN_TransformIntoDisplayableImage : Node_F_VN_TransformIntoDisplayableImage;
    node_F_VN_TransformIntoDisplayableImageExp : Node_F_VN_TransformIntoDisplayableImageExp;
    node_F_VN_CreateNDimensionalImage : Node_F_VN_CreateNDimensionalImage;
    node_F_VN_CreateNDimensionalImageAndSetPixels : Node_F_VN_CreateNDimensionalImageAndSetPixels;
    //node_F_VN_CreateNDimensionalImageFromArray : Node_F_VN_CreateNDimensionalImageFromArray;
    node_F_VN_GetLayoutInfo : Node_F_VN_GetLayoutInfo;
    node_F_VN_PadImageBorder : Node_F_VN_PadImageBorder;
    node_F_VN_PadImageBorderExp : Node_F_VN_PadImageBorderExp;
    //node_F_VN_ReinterpretUnsupportedImage : Node_F_VN_ReinterpretUnsupportedImage;
    
    // Code Quality
    node_F_VN_GradeBarcode : Node_F_VN_GradeBarcode;
    node_F_VN_GradeBarcodeExp : Node_F_VN_GradeBarcodeExp;
    node_F_VN_GradeDataMatrixCode : Node_F_VN_GradeDataMatrixCode;
    node_F_VN_GradeDataMatrixCodeExp : Node_F_VN_GradeDataMatrixCodeExp;
    node_F_VN_GradeQRCode : Node_F_VN_GradeQRCode;
    node_F_VN_GradeQRCodeExp : Node_F_VN_GradeQRCodeExp;
    
    // Code Reading
    node_F_VN_AnalyzeBarcodeWalsh : Node_F_VN_AnalyzeBarcodeWalsh;
    node_F_VN_DetectBarcodesWalsh : Node_F_VN_DetectBarcodesWalsh;
	node_F_VN_DetectCodesNeuralNetwork : Node_F_VN_DetectCodesNeuralNetwork;
    node_F_VN_ReadBarcode : Node_F_VN_ReadBarcode;
	node_F_VN_ReadBarcodeExp : Node_F_VN_ReadBarcodeExp;
	node_F_VN_ReadBarcodeExp2 : Node_F_VN_ReadBarcodeExp2;
    node_F_VN_ReadBarcodeRoi : Node_F_VN_ReadBarcodeRoi;
    node_F_VN_ReadBarcodeRoiExp : Node_F_VN_ReadBarcodeRoiExp;
    node_F_VN_ReadDataMatrixCode : Node_F_VN_ReadDataMatrixCode;
	node_F_VN_ReadDataMatrixCodeExp : Node_F_VN_ReadDataMatrixCodeExp;
	node_F_VN_ReadDataMatrixCodeExp2 : Node_F_VN_ReadDataMatrixCodeExp2;
	node_F_VN_ReadDataMatrixCodeRoi : Node_F_VN_ReadDataMatrixCodeRoi;
    node_F_VN_ReadDataMatrixCodeRoiExp : Node_F_VN_ReadDataMatrixCodeRoiExp;
	node_F_VN_ReadDotCodeRoi : Node_F_VN_ReadDotCodeRoi;
	node_F_VN_ReadDotCodeRoiExp : Node_F_VN_ReadDotCodeRoiExp;
    node_F_VN_ReadPharmaCode : Node_F_VN_ReadPharmaCode;
	node_F_VN_ReadPharmaCodeExp : Node_F_VN_ReadPharmaCodeExp;
	node_F_VN_ReadPharmaCodeExp2 : Node_F_VN_ReadPharmaCodeExp2;
    node_F_VN_ReadQRCode : Node_F_VN_ReadQRCode;
	node_F_VN_ReadQRCodeExp : Node_F_VN_ReadQRCodeExp;
	node_F_VN_ReadQRCodeExp2 : Node_F_VN_ReadQRCodeExp2;
    
    // Constants
    node_RGBA_BLACK : Node_RGBA_BLACK;
    node_RGBA_RED : Node_RGBA_RED;
    node_RGBA_YELLOW : Node_RGBA_YELLOW;
    node_RGBA_GREEN : Node_RGBA_GREEN;
    node_RGBA_CYAN : Node_RGBA_CYAN;
    node_RGBA_BLUE : Node_RGBA_BLUE;
    node_RGBA_MAGENTA : Node_RGBA_MAGENTA;
    node_RGBA_WHITE : Node_RGBA_WHITE;
    node_RGBA_RANDOM : Node_RGBA_RANDOM;
	node_ContainerType_Vector_SINT : Node_ContainerType_Vector_SINT;
	node_ContainerType_Vector_USINT : Node_ContainerType_Vector_USINT;
	node_ContainerType_Vector_INT : Node_ContainerType_Vector_INT;
	node_ContainerType_Vector_UINT : Node_ContainerType_Vector_UINT;
	node_ContainerType_Vector_DINT : Node_ContainerType_Vector_DINT;
	node_ContainerType_Vector_UDINT : Node_ContainerType_Vector_UDINT;
	node_ContainerType_Vector_ULINT : Node_ContainerType_Vector_ULINT;
	node_ContainerType_Vector_REAL : Node_ContainerType_Vector_REAL;
	node_ContainerType_Vector_LREAL : Node_ContainerType_Vector_LREAL;
	node_ContainerType_Vector_ITcVnImage : Node_ContainerType_Vector_ITcVnImage;
	node_ContainerType_Vector_TcVnPoint2_DINT : Node_ContainerType_Vector_TcVnPoint2_DINT;
	node_ContainerType_Vector_TcVnPoint2_REAL : Node_ContainerType_Vector_TcVnPoint2_REAL;
	node_ContainerType_Vector_TcVnPoint2_LREAL : Node_ContainerType_Vector_TcVnPoint2_LREAL;
	node_ContainerType_Vector_TcVnPoint3_REAL : Node_ContainerType_Vector_TcVnPoint3_REAL;
	node_ContainerType_Vector_TcVnPoint3_LREAL : Node_ContainerType_Vector_TcVnPoint3_LREAL;
	node_ContainerType_Vector_Vector_TcVnPoint2_DINT : Node_ContainerType_Vector_Vector_TcVnPoint2_DINT;
	node_ContainerType_Vector_Vector_TcVnPoint2_REAL : Node_ContainerType_Vector_Vector_TcVnPoint2_REAL;
	node_ContainerType_Vector_Vector_TcVnPoint3_REAL : Node_ContainerType_Vector_Vector_TcVnPoint3_REAL;
	node_ContainerType_Vector_Vector_UDINT : Node_ContainerType_Vector_Vector_UDINT;
	node_ContainerType_Vector_Vector_ULINT : Node_ContainerType_Vector_Vector_ULINT;
	node_ContainerType_Vector_Vector_REAL : Node_ContainerType_Vector_Vector_REAL;
	node_ContainerType_Vector_Vector_LREAL : Node_ContainerType_Vector_Vector_LREAL;
	node_ContainerType_Vector_TcVnVector2_SINT : Node_ContainerType_Vector_TcVnVector2_SINT;
	node_ContainerType_Vector_TcVnVector2_USINT : Node_ContainerType_Vector_TcVnVector2_USINT;
	node_ContainerType_Vector_TcVnVector2_INT : Node_ContainerType_Vector_TcVnVector2_INT;
	node_ContainerType_Vector_TcVnVector2_UINT : Node_ContainerType_Vector_TcVnVector2_UINT;
	node_ContainerType_Vector_TcVnVector2_DINT : Node_ContainerType_Vector_TcVnVector2_DINT;
	node_ContainerType_Vector_TcVnVector2_REAL : Node_ContainerType_Vector_TcVnVector2_REAL;
	node_ContainerType_Vector_TcVnVector3_SINT : Node_ContainerType_Vector_TcVnVector3_SINT;
	node_ContainerType_Vector_TcVnVector3_USINT : Node_ContainerType_Vector_TcVnVector3_USINT;
	node_ContainerType_Vector_TcVnVector3_INT : Node_ContainerType_Vector_TcVnVector3_INT;
	node_ContainerType_Vector_TcVnVector3_UINT : Node_ContainerType_Vector_TcVnVector3_UINT;
	node_ContainerType_Vector_TcVnVector3_REAL : Node_ContainerType_Vector_TcVnVector3_REAL;
	node_ContainerType_Vector_TcVnVector4_SINT : Node_ContainerType_Vector_TcVnVector4_SINT;
	node_ContainerType_Vector_TcVnVector4_USINT : Node_ContainerType_Vector_TcVnVector4_USINT;
	node_ContainerType_Vector_TcVnVector4_INT : Node_ContainerType_Vector_TcVnVector4_INT;
	node_ContainerType_Vector_TcVnVector4_UINT : Node_ContainerType_Vector_TcVnVector4_UINT;
	node_ContainerType_Vector_TcVnVector4_DINT : Node_ContainerType_Vector_TcVnVector4_DINT;
	node_ContainerType_Vector_TcVnVector4_REAL : Node_ContainerType_Vector_TcVnVector4_REAL;
	node_ContainerType_Vector_TcVnVector4_LREAL : Node_ContainerType_Vector_TcVnVector4_LREAL;
	node_ContainerType_Vector_TcVnRectangle_DINT : Node_ContainerType_Vector_TcVnRectangle_DINT;
	node_ContainerType_Vector_TcVnRotatedRectangle : Node_ContainerType_Vector_TcVnRotatedRectangle;
	node_ContainerType_Vector_TcVnKeyPoint : Node_ContainerType_Vector_TcVnKeyPoint;
	node_ContainerType_Vector_TcVnDMatch : Node_ContainerType_Vector_TcVnDMatch;
	node_ContainerType_Vector_Vector_TcVnDMatch : Node_ContainerType_Vector_Vector_TcVnDMatch;
	node_ContainerType_String_SINT : Node_ContainerType_String_SINT;
	node_ContainerType_Vector_String_SINT : Node_ContainerType_Vector_String_SINT;
    
    // Container Statistics
    node_F_VN_MaxElementElementwise_DINT : Node_F_VN_MaxElementElementwise_DINT;
    node_F_VN_MaxElementElementwise_INT : Node_F_VN_MaxElementElementwise_INT;
    node_F_VN_MaxElementElementwise_LREAL : Node_F_VN_MaxElementElementwise_LREAL;
    node_F_VN_MaxElementElementwise_REAL : Node_F_VN_MaxElementElementwise_REAL;
    node_F_VN_MaxElementElementwise_SINT : Node_F_VN_MaxElementElementwise_SINT;
    node_F_VN_MaxElementElementwise_TcVnPoint2_DINT : Node_F_VN_MaxElementElementwise_TcVnPoint2_DINT;
    node_F_VN_MaxElementElementwise_TcVnPoint2_LREAL : Node_F_VN_MaxElementElementwise_TcVnPoint2_LREAL;
    node_F_VN_MaxElementElementwise_TcVnPoint2_REAL : Node_F_VN_MaxElementElementwise_TcVnPoint2_REAL;
    node_F_VN_MaxElementElementwise_TcVnPoint3_LREAL : Node_F_VN_MaxElementElementwise_TcVnPoint3_LREAL;
    node_F_VN_MaxElementElementwise_TcVnPoint3_REAL : Node_F_VN_MaxElementElementwise_TcVnPoint3_REAL;
    node_F_VN_MaxElementElementwise_TcVnVector2_DINT : Node_F_VN_MaxElementElementwise_TcVnVector2_DINT;
    node_F_VN_MaxElementElementwise_TcVnVector2_INT : Node_F_VN_MaxElementElementwise_TcVnVector2_INT;
    node_F_VN_MaxElementElementwise_TcVnVector2_REAL : Node_F_VN_MaxElementElementwise_TcVnVector2_REAL;
    node_F_VN_MaxElementElementwise_TcVnVector2_SINT : Node_F_VN_MaxElementElementwise_TcVnVector2_SINT;
    node_F_VN_MaxElementElementwise_TcVnVector2_UINT : Node_F_VN_MaxElementElementwise_TcVnVector2_UINT;
    node_F_VN_MaxElementElementwise_TcVnVector2_USINT : Node_F_VN_MaxElementElementwise_TcVnVector2_USINT;
    node_F_VN_MaxElementElementwise_TcVnVector3_INT : Node_F_VN_MaxElementElementwise_TcVnVector3_INT;
    node_F_VN_MaxElementElementwise_TcVnVector3_REAL : Node_F_VN_MaxElementElementwise_TcVnVector3_REAL;
    node_F_VN_MaxElementElementwise_TcVnVector3_SINT : Node_F_VN_MaxElementElementwise_TcVnVector3_SINT;
    node_F_VN_MaxElementElementwise_TcVnVector3_UINT : Node_F_VN_MaxElementElementwise_TcVnVector3_UINT;
    node_F_VN_MaxElementElementwise_TcVnVector3_USINT : Node_F_VN_MaxElementElementwise_TcVnVector3_USINT;
    node_F_VN_MaxElementElementwise_TcVnVector4_DINT : Node_F_VN_MaxElementElementwise_TcVnVector4_DINT;
    node_F_VN_MaxElementElementwise_TcVnVector4_INT : Node_F_VN_MaxElementElementwise_TcVnVector4_INT;
    node_F_VN_MaxElementElementwise_TcVnVector4_LREAL : Node_F_VN_MaxElementElementwise_TcVnVector4_LREAL;
    node_F_VN_MaxElementElementwise_TcVnVector4_REAL : Node_F_VN_MaxElementElementwise_TcVnVector4_REAL;
    node_F_VN_MaxElementElementwise_TcVnVector4_SINT : Node_F_VN_MaxElementElementwise_TcVnVector4_SINT;
    node_F_VN_MaxElementElementwise_TcVnVector4_UINT : Node_F_VN_MaxElementElementwise_TcVnVector4_UINT;
    node_F_VN_MaxElementElementwise_TcVnVector4_USINT : Node_F_VN_MaxElementElementwise_TcVnVector4_USINT;
    node_F_VN_MaxElementElementwise_UDINT : Node_F_VN_MaxElementElementwise_UDINT;
    node_F_VN_MaxElementElementwise_UINT : node_F_VN_MaxElementElementwise_UINT;
    node_F_VN_MaxElementElementwise_ULINT : Node_F_VN_MaxElementElementwise_ULINT;
    node_F_VN_MaxElementElementwise_USINT : Node_F_VN_MaxElementElementwise_USINT;
    node_F_VN_MedianElementElementwise_DINT : Node_F_VN_MedianElementElementwise_DINT;
    node_F_VN_MedianElementElementwise_INT : Node_F_VN_MedianElementElementwise_INT;
    node_F_VN_MedianElementElementwise_LREAL : Node_F_VN_MedianElementElementwise_LREAL;
    node_F_VN_MedianElementElementwise_REAL : Node_F_VN_MedianElementElementwise_REAL;
    node_F_VN_MedianElementElementwise_SINT : Node_F_VN_MedianElementElementwise_SINT;
    node_F_VN_MedianElementElementwise_TcVnPoint2_DINT : Node_F_VN_MedianElementElementwise_TcVnPoint2_DINT;
    node_F_VN_MedianElementElementwise_TcVnPoint2_LREAL : Node_F_VN_MedianElementElementwise_TcVnPoint2_LREAL;
    node_F_VN_MedianElementElementwise_TcVnPoint2_REAL : Node_F_VN_MedianElementElementwise_TcVnPoint2_REAL;
    node_F_VN_MedianElementElementwise_TcVnPoint3_LREAL : Node_F_VN_MedianElementElementwise_TcVnPoint3_LREAL;
    node_F_VN_MedianElementElementwise_TcVnPoint3_REAL : Node_F_VN_MedianElementElementwise_TcVnPoint3_REAL;
    node_F_VN_MedianElementElementwise_TcVnVector2_DINT : Node_F_VN_MedianElementElementwise_TcVnVector2_DINT;
    node_F_VN_MedianElementElementwise_TcVnVector2_INT : Node_F_VN_MedianElementElementwise_TcVnVector2_INT;
    node_F_VN_MedianElementElementwise_TcVnVector2_REAL : Node_F_VN_MedianElementElementwise_TcVnVector2_REAL;
    node_F_VN_MedianElementElementwise_TcVnVector2_SINT : Node_F_VN_MedianElementElementwise_TcVnVector2_SINT;
    node_F_VN_MedianElementElementwise_TcVnVector2_UINT : Node_F_VN_MedianElementElementwise_TcVnVector2_UINT;
    node_F_VN_MedianElementElementwise_TcVnVector2_USINT : Node_F_VN_MedianElementElementwise_TcVnVector2_USINT;
    node_F_VN_MedianElementElementwise_TcVnVector3_INT : Node_F_VN_MedianElementElementwise_TcVnVector3_INT;
    node_F_VN_MedianElementElementwise_TcVnVector3_REAL : Node_F_VN_MedianElementElementwise_TcVnVector3_REAL;
    node_F_VN_MedianElementElementwise_TcVnVector3_SINT : Node_F_VN_MedianElementElementwise_TcVnVector3_SINT;
    node_F_VN_MedianElementElementwise_TcVnVector3_UINT : Node_F_VN_MedianElementElementwise_TcVnVector3_UINT;
    node_F_VN_MedianElementElementwise_TcVnVector3_USINT : Node_F_VN_MedianElementElementwise_TcVnVector3_USINT;
    node_F_VN_MedianElementElementwise_TcVnVector4_DINT : Node_F_VN_MedianElementElementwise_TcVnVector4_DINT;
    node_F_VN_MedianElementElementwise_TcVnVector4_INT : Node_F_VN_MedianElementElementwise_TcVnVector4_INT;
    node_F_VN_MedianElementElementwise_TcVnVector4_LREAL : Node_F_VN_MedianElementElementwise_TcVnVector4_LREAL;
    node_F_VN_MedianElementElementwise_TcVnVector4_REAL : Node_F_VN_MedianElementElementwise_TcVnVector4_REAL;
    node_F_VN_MedianElementElementwise_TcVnVector4_SINT : Node_F_VN_MedianElementElementwise_TcVnVector4_SINT;
    node_F_VN_MedianElementElementwise_TcVnVector4_UINT : Node_F_VN_MedianElementElementwise_TcVnVector4_UINT;
    node_F_VN_MedianElementElementwise_TcVnVector4_USINT : Node_F_VN_MedianElementElementwise_TcVnVector4_USINT;
    node_F_VN_MedianElementElementwise_UDINT : Node_F_VN_MedianElementElementwise_UDINT;
    node_F_VN_MedianElementElementwise_UINT : node_F_VN_MedianElementElementwise_UINT;
    node_F_VN_MedianElementElementwise_ULINT : Node_F_VN_MedianElementElementwise_ULINT;
    node_F_VN_MedianElementElementwise_USINT : Node_F_VN_MedianElementElementwise_USINT;
    node_F_VN_MinElementElementwise_DINT : Node_F_VN_MinElementElementwise_DINT;
    node_F_VN_MinElementElementwise_INT : Node_F_VN_MinElementElementwise_INT;
    node_F_VN_MinElementElementwise_LREAL : Node_F_VN_MinElementElementwise_LREAL;
    node_F_VN_MinElementElementwise_REAL : Node_F_VN_MinElementElementwise_REAL;
    node_F_VN_MinElementElementwise_SINT : Node_F_VN_MinElementElementwise_SINT;
    node_F_VN_MinElementElementwise_TcVnPoint2_DINT : Node_F_VN_MinElementElementwise_TcVnPoint2_DINT;
    node_F_VN_MinElementElementwise_TcVnPoint2_LREAL : Node_F_VN_MinElementElementwise_TcVnPoint2_LREAL;
    node_F_VN_MinElementElementwise_TcVnPoint2_REAL : Node_F_VN_MinElementElementwise_TcVnPoint2_REAL;
    node_F_VN_MinElementElementwise_TcVnPoint3_LREAL : Node_F_VN_MinElementElementwise_TcVnPoint3_LREAL;
    node_F_VN_MinElementElementwise_TcVnPoint3_REAL : Node_F_VN_MinElementElementwise_TcVnPoint3_REAL;
    node_F_VN_MinElementElementwise_TcVnVector2_DINT : Node_F_VN_MinElementElementwise_TcVnVector2_DINT;
    node_F_VN_MinElementElementwise_TcVnVector2_INT : Node_F_VN_MinElementElementwise_TcVnVector2_INT;
    node_F_VN_MinElementElementwise_TcVnVector2_REAL : Node_F_VN_MinElementElementwise_TcVnVector2_REAL;
    node_F_VN_MinElementElementwise_TcVnVector2_SINT : Node_F_VN_MinElementElementwise_TcVnVector2_SINT;
    node_F_VN_MinElementElementwise_TcVnVector2_UINT : Node_F_VN_MinElementElementwise_TcVnVector2_UINT;
    node_F_VN_MinElementElementwise_TcVnVector2_USINT : Node_F_VN_MinElementElementwise_TcVnVector2_USINT;
    node_F_VN_MinElementElementwise_TcVnVector3_INT : Node_F_VN_MinElementElementwise_TcVnVector3_INT;
    node_F_VN_MinElementElementwise_TcVnVector3_REAL : Node_F_VN_MinElementElementwise_TcVnVector3_REAL;
    node_F_VN_MinElementElementwise_TcVnVector3_SINT : Node_F_VN_MinElementElementwise_TcVnVector3_SINT;
    node_F_VN_MinElementElementwise_TcVnVector3_UINT : Node_F_VN_MinElementElementwise_TcVnVector3_UINT;
    node_F_VN_MinElementElementwise_TcVnVector3_USINT : Node_F_VN_MinElementElementwise_TcVnVector3_USINT;
    node_F_VN_MinElementElementwise_TcVnVector4_DINT : Node_F_VN_MinElementElementwise_TcVnVector4_DINT;
    node_F_VN_MinElementElementwise_TcVnVector4_INT : Node_F_VN_MinElementElementwise_TcVnVector4_INT;
    node_F_VN_MinElementElementwise_TcVnVector4_LREAL : Node_F_VN_MinElementElementwise_TcVnVector4_LREAL;
    node_F_VN_MinElementElementwise_TcVnVector4_REAL : Node_F_VN_MinElementElementwise_TcVnVector4_REAL;
    node_F_VN_MinElementElementwise_TcVnVector4_SINT : Node_F_VN_MinElementElementwise_TcVnVector4_SINT;
    node_F_VN_MinElementElementwise_TcVnVector4_UINT : Node_F_VN_MinElementElementwise_TcVnVector4_UINT;
    node_F_VN_MinElementElementwise_TcVnVector4_USINT : Node_F_VN_MinElementElementwise_TcVnVector4_USINT;
    node_F_VN_MinElementElementwise_UDINT : Node_F_VN_MinElementElementwise_UDINT;
    node_F_VN_MinElementElementwise_UINT : node_F_VN_MinElementElementwise_UINT;
    node_F_VN_MinElementElementwise_ULINT : Node_F_VN_MinElementElementwise_ULINT;
    node_F_VN_MinElementElementwise_USINT : Node_F_VN_MinElementElementwise_USINT;
	node_F_VN_ContainerAverage : Node_F_VN_ContainerAverage;
	node_F_VN_ContainerAverageElementwise2 : Node_F_VN_ContainerAverageElementwise2;
	node_F_VN_ContainerAverageElementwise3 : Node_F_VN_ContainerAverageElementwise3;
	node_F_VN_ContainerAverageElementwise4 : Node_F_VN_ContainerAverageElementwise4;
	node_F_VN_ContainerAverageVariance : Node_F_VN_ContainerAverageVariance;
	node_F_VN_ContainerAverageVarianceElementwise2 : Node_F_VN_ContainerAverageVarianceElementwise2;
	node_F_VN_ContainerAverageVarianceElementwise3 : Node_F_VN_ContainerAverageVarianceElementwise3;
	node_F_VN_ContainerAverageVarianceElementwise4 : Node_F_VN_ContainerAverageVarianceElementwise4;
	node_F_VN_MaxElement : Node_F_VN_MaxElement;
	node_F_VN_MedianElement : Node_F_VN_MedianElement;
	node_F_VN_MinElement : Node_F_VN_MinElement;
   
    // Contour Analysis
    node_F_VN_ApproximatePolygon : Node_F_VN_ApproximatePolygon;
    node_F_VN_CheckIfPointIsInsideContour : Node_F_VN_CheckIfPointIsInsideContour;
    node_F_VN_ContourArea : Node_F_VN_ContourArea;
    node_F_VN_ContourCenterOfMass : Node_F_VN_ContourCenterOfMass;
    node_F_VN_ContourCircularity : Node_F_VN_ContourCircularity;
    node_F_VN_ContourCircularityExp : Node_F_VN_ContourCircularityExp;
    node_F_VN_ContourConvexity : Node_F_VN_ContourConvexity;
    node_F_VN_ContourEccentricity : Node_F_VN_ContourEccentricity;
    node_F_VN_ContourElongation : Node_F_VN_ContourElongation;
    node_F_VN_ContourExtremePoint : Node_F_VN_ContourExtremePoint;
    node_F_VN_ContourInertiaRatio : Node_F_VN_ContourInertiaRatio;
    node_F_VN_ContourMoments : Node_F_VN_ContourMoments;
    node_F_VN_ContourOrientation : Node_F_VN_ContourOrientation;
    node_F_VN_ContourOrientationExp : Node_F_VN_ContourOrientationExp;
    node_F_VN_ContourPerimeter : Node_F_VN_ContourPerimeter;
    node_F_VN_ContourRoundness : Node_F_VN_ContourRoundness;
    node_F_VN_ConvexHullPoints : Node_F_VN_ConvexHullPoints;
    node_F_VN_ConvexHullPointsExp : Node_F_VN_ConvexHullPointsExp;
    node_F_VN_ConvexityDefects : Node_F_VN_ConvexityDefects;
    //node_F_VN_CustomElementWiseContainerOperation_ITcVnContainer : Node_F_VN_CustomElementWiseContainerOperation_ITcVnContainer;
    //node_F_VN_CustomElementWiseContainerOperation_ITcVnForwardIterator : Node_F_VN_CustomElementWiseContainerOperation_ITcVnForwardIterator;
    node_F_VN_EnclosingCircle : Node_F_VN_EnclosingCircle;
    node_F_VN_EnclosingRectangle : Node_F_VN_EnclosingRectangle;
    node_F_VN_EnclosingTriangle : Node_F_VN_EnclosingTriangle;
    node_F_VN_FitEllipse : Node_F_VN_FitEllipse;
    node_F_VN_FitLine : Node_F_VN_FitLine;
	node_F_VN_FitLineExp : Node_F_VN_FitLineExp;
    //node_F_VN_FourierDescriptors : Node_F_VN_FourierDescriptors;
    node_F_VN_MatchContours : Node_F_VN_MatchContours;
    node_F_VN_MatchContours1vsN : Node_F_VN_MatchContours1vsN;
    node_F_VN_MatchContours1vsNExp : Node_F_VN_MatchContours1vsNExp;
    node_F_VN_MatchContoursExp : Node_F_VN_MatchContoursExp;
    node_F_VN_UprightBoundingRectangle : Node_F_VN_UprightBoundingRectangle;
    
    // Control Functions
    //node_F_VN_StartAbsWatchdog : Node_F_VN_StartAbsWatchdog;
    //node_F_VN_StartAbsWatchdogExp : Node_F_VN_StartAbsWatchdogExp;
    //node_F_VN_StartRelWatchdog : Node_F_VN_StartRelWatchdog;
    //node_F_VN_StartRelWatchdogExp : Node_F_VN_StartRelWatchdogExp;
    //node_F_VN_StopWatchdog : Node_F_VN_StopWatchdog;
    
    // Drawing
    node_F_VN_DrawArrow : Node_F_VN_DrawArrow;
    node_F_VN_DrawArrow_TcVnVector4_DINT : Node_F_VN_DrawArrow_TcVnVector4_DINT;
    node_F_VN_DrawArrowExp : Node_F_VN_DrawArrowExp;
    node_F_VN_DrawArrowExp_TcVnVector4_DINT : Node_F_VN_DrawArrowExp_TcVnVector4_DINT;
    node_F_VN_DrawCircle : Node_F_VN_DrawCircle;
    node_F_VN_DrawCircleExp : Node_F_VN_DrawCircleExp;
    node_F_VN_DrawCircles : Node_F_VN_DrawCircles;
    node_F_VN_DrawCirclesExp : Node_F_VN_DrawCirclesExp;
    node_F_VN_DrawCircularArc : Node_F_VN_DrawCircularArc;
    node_F_VN_DrawCircularArcExp : Node_F_VN_DrawCircularArcExp;
    node_F_VN_DrawComponents : Node_F_VN_DrawComponents;
    node_F_VN_DrawComponentsExp : Node_F_VN_DrawComponentsExp;
    node_F_VN_DrawContours : Node_F_VN_DrawContours;
    node_F_VN_DrawContoursExp : Node_F_VN_DrawContoursExp;
    node_F_VN_DrawEllipse : Node_F_VN_DrawEllipse;
    node_F_VN_DrawEllipseExp : Node_F_VN_DrawEllipseExp;
    node_F_VN_DrawKeypoints : Node_F_VN_DrawKeypoints;
    node_F_VN_DrawKeypointsExp : Node_F_VN_DrawKeypointsExp;
    node_F_VN_DrawLine : Node_F_VN_DrawLine;
    node_F_VN_DrawLine_TcVnVector4_DINT : Node_F_VN_DrawLine_TcVnVector4_DINT;
    node_F_VN_DrawLine_TcVnVector4_LREAL : Node_F_VN_DrawLine_TcVnVector4_LREAL;
    node_F_VN_DrawLineExp : Node_F_VN_DrawLineExp;
    node_F_VN_DrawLineExp_TcVnVector4_DINT : Node_F_VN_DrawLineExp_TcVnVector4_DINT;
    node_F_VN_DrawLineExp_TcVnVector4_LREAL : Node_F_VN_DrawLineExp_TcVnVector4_LREAL;
    node_F_VN_DrawLines : Node_F_VN_DrawLines;
    node_F_VN_DrawLinesExp : Node_F_VN_DrawLinesExp;
    node_F_VN_DrawMatches : Node_F_VN_DrawMatches;
    node_F_VN_DrawMatchesExp : Node_F_VN_DrawMatchesExp;
    node_F_VN_DrawOrientation : Node_F_VN_DrawOrientation;
    node_F_VN_DrawOrientationExp : Node_F_VN_DrawOrientationExp;
    node_F_VN_DrawPoint : Node_F_VN_DrawPoint;
    node_F_VN_DrawPointExp : Node_F_VN_DrawPointExp;
    node_F_VN_DrawPoints : Node_F_VN_DrawPoints;
    node_F_VN_DrawPointsExp : Node_F_VN_DrawPointsExp;
    node_F_VN_DrawPolygon : Node_F_VN_DrawPolygon;
    node_F_VN_DrawPolygonExp : Node_F_VN_DrawPolygonExp;
    node_F_VN_DrawRectangle : Node_F_VN_DrawRectangle;
    node_F_VN_DrawRectangle_TcVnRectangle_DINT : Node_F_VN_DrawRectangle_TcVnRectangle_DINT;
    node_F_VN_DrawRectangle_TcVnRectangle_UDINT : Node_F_VN_DrawRectangle_TcVnRectangle_UDINT;
    node_F_VN_DrawRotatedRectangle : Node_F_VN_DrawRotatedRectangle;
    node_F_VN_DrawRotatedRectangleExp : Node_F_VN_DrawRotatedRectangleExp;
    node_F_VN_FillCircle : Node_F_VN_FillCircle;
    node_F_VN_FillContours : Node_F_VN_FillContours;
    node_F_VN_FillEllipse : Node_F_VN_FillEllipse;
    node_F_VN_FillPolygon : Node_F_VN_FillPolygon;
    node_F_VN_FillRectangle : Node_F_VN_FillRectangle;
    node_F_VN_FillRotatedRectangle : Node_F_VN_FillRotatedRectangle;
    node_F_VN_PlotIntensityProfile : Node_F_VN_PlotIntensityProfile;
    node_F_VN_PlotIntensityProfileExp : Node_F_VN_PlotIntensityProfileExp;
    node_F_VN_PutLabel : Node_F_VN_PutLabel;
    node_F_VN_PutLabelExp : Node_F_VN_PutLabelExp;
    node_F_VN_PutText : Node_F_VN_PutText;
    node_F_VN_PutTextExp : Node_F_VN_PutTextExp;
    
    // Fourier Analysis
    node_F_VN_CreateBandpassButterworthFilter : Node_F_VN_CreateBandpassButterworthFilter;
    node_F_VN_CreateBandpassGaussianFilter : Node_F_VN_CreateBandpassGaussianFilter;
    node_F_VN_CreateBandrejectButterworthFilter : Node_F_VN_CreateBandrejectButterworthFilter;
    node_F_VN_CreateBandrejectGaussianFilter : Node_F_VN_CreateBandrejectGaussianFilter;
    node_F_VN_CreateHighpassButterworthFilter : Node_F_VN_CreateHighpassButterworthFilter;
    node_F_VN_CreateHighpassGaussianFilter : Node_F_VN_CreateHighpassGaussianFilter;
    node_F_VN_CreateLowpassButterworthFilter : Node_F_VN_CreateLowpassButterworthFilter;
    node_F_VN_CreateLowpassGaussianFilter : Node_F_VN_CreateLowpassGaussianFilter;
    node_F_VN_Dft : Node_F_VN_Dft;
    node_F_VN_InverseDft : Node_F_VN_InverseDft;
    node_F_VN_OptimalDftSize : Node_F_VN_OptimalDftSize;
    
